C07284=1024.392,-31.797,405.502,166.984,47.714,158.740
C07285=1024.386,-32.047,405.514,166.981,47.718,158.740
C07286=1024.380,-32.296,405.527,166.978,47.721,158.740
C07287=1024.374,-32.546,405.540,166.975,47.724,158.741
C07288=1024.368,-32.796,405.553,166.973,47.727,158.741
C07289=1024.362,-33.046,405.565,166.970,47.731,158.741
C07290=1024.356,-33.295,405.578,166.967,47.734,158.741
C07291=1024.350,-33.545,405.590,166.964,47.737,158.741
C07292=1024.344,-33.794,405.603,166.961,47.740,158.742
C07293=1024.338,-34.044,405.615,166.958,47.744,158.742
C07294=1024.332,-34.293,405.628,166.955,47.747,158.742
C07295=1024.326,-34.543,405.641,166.953,47.750,158.742
C07296=1024.320,-34.793,405.653,166.950,47.753,158.742
C07297=1024.314,-35.043,405.666,166.947,47.757,158.743
C07298=1024.308,-35.292,405.679,166.945,47.760,158.743
C07299=1024.303,-35.541,405.691,166.942,47.763,158.743
C07300=1024.296,-35.791,405.703,166.938,47.766,158.743
C07301=1024.290,-36.040,405.716,166.935,47.770,158.743
C07302=1024.284,-36.290,405.729,166.933,47.772,158.744
C07303=1024.278,-36.570,405.743,166.930,47.776,158.744
C07304=1024.272,-36.849,405.757,166.926,47.780,158.744
C07305=1024.265,-37.129,405.770,166.923,47.784,158.744
C07306=1024.258,-37.408,405.785,166.920,47.787,158.745
C07307=1024.252,-37.658,405.797,166.917,47.791,158.745
C07308=1024.246,-37.908,405.810,166.915,47.793,158.745
C07309=1024.241,-38.157,405.822,166.912,47.797,158.745
C07310=1024.234,-38.407,405.834,166.908,47.800,158.745
C07311=1024.228,-38.656,405.847,166.905,47.803,158.745
C07312=1024.222,-38.906,405.860,166.903,47.807,158.746
C07313=1024.216,-39.156,405.872,166.900,47.810,158.746
C07314=1024.211,-39.405,405.885,166.897,47.813,158.746
C07315=1024.204,-39.654,405.897,166.894,47.816,158.746
C07316=1024.198,-39.904,405.909,166.892,47.820,158.747
C07317=1024.193,-40.155,405.921,166.889,47.823,158.747
C07318=1024.187,-40.404,405.933,166.886,47.826,158.747
C07319=1024.181,-40.654,405.945,166.883,47.830,158.747
C07320=1024.175,-40.903,405.958,166.880,47.833,158.747
C07321=1024.168,-41.153,405.970,166.877,47.836,158.748
C07322=1024.163,-41.402,405.982,166.874,47.840,158.748
C07323=1024.156,-41.652,405.994,166.871,47.843,158.748
C07324=1024.151,-41.902,406.006,166.868,47.846,158.748
C07325=1024.145,-42.152,406.019,166.866,47.850,158.748
C07326=1024.139,-42.400,406.031,166.863,47.853,158.749
C07327=1024.133,-42.650,406.043,166.860,47.856,158.749
C07328=1024.126,-42.900,406.054,166.857,47.859,158.749
C07329=1024.121,-43.150,406.067,166.854,47.863,158.749
C07330=1024.115,-43.400,406.079,166.852,47.866,158.749
C07331=1024.108,-43.649,406.091,166.848,47.869,158.750
C07332=1024.103,-43.899,406.104,166.845,47.873,158.750
C07333=1024.097,-44.148,406.115,166.842,47.876,158.750
C07334=1024.091,-44.398,406.128,166.839,47.879,158.750
C07335=1024.085,-44.648,406.140,166.837,47.882,158.750
C07336=1024.079,-44.897,406.151,166.834,47.886,158.751
C07337=1024.073,-45.147,406.164,166.831,47.889,158.751
C07338=1024.067,-45.396,406.175,166.828,47.892,158.751
C07339=1024.061,-45.646,406.188,166.825,47.895,158.751
C07340=1024.055,-45.896,406.200,166.823,47.899,158.751
C07341=1024.049,-46.145,406.211,166.819,47.902,158.752
C07342=1024.044,-46.395,406.224,166.816,47.905,158.752
C07343=1024.037,-46.645,406.236,166.813,47.909,158.752
C07344=1024.032,-46.894,406.247,166.811,47.912,158.752
C07345=1024.026,-47.144,406.260,166.808,47.915,158.752
C07346=1024.020,-47.393,406.271,166.805,47.918,158.753
C07347=1024.014,-47.643,406.284,166.802,47.922,158.753
C07348=1024.008,-47.893,406.295,166.799,47.925,158.753
C07349=1024.002,-48.142,406.307,166.797,47.928,158.753
C07350=1023.996,-48.392,406.320,166.793,47.932,158.753
C07351=1023.991,-48.642,406.331,166.790,47.935,158.753
C07352=1023.985,-48.892,406.343,166.787,47.938,158.754
C07353=1023.978,-49.141,406.355,166.785,47.941,158.754
C07354=1023.973,-49.391,406.367,166.782,47.945,158.754
C07355=1023.967,-49.641,406.379,166.779,47.948,158.754
C07356=1023.961,-49.890,406.391,166.776,47.951,158.754
C07357=1023.956,-50.140,406.403,166.773,47.954,158.755
C07358=1023.950,-50.389,406.414,166.770,47.957,158.755
C07359=1023.944,-50.639,406.427,166.767,47.961,158.755
C07360=1023.938,-50.889,406.438,166.764,47.964,158.755
C07361=1023.931,-51.138,406.450,166.761,47.967,158.755
C07362=1023.926,-51.389,406.462,166.758,47.971,158.756
C07363=1023.920,-51.637,406.473,166.755,47.974,158.756
C07364=1023.913,-51.888,406.484,166.753,47.978,158.756
C07365=1023.908,-52.137,406.495,166.750,47.981,158.756
C07366=1023.901,-52.387,406.507,166.747,47.984,158.756
C07367=1023.894,-52.666,406.520,166.743,47.988,158.757
C07368=1023.887,-52.947,406.533,166.740,47.992,158.757
C07369=1023.881,-53.227,406.546,166.737,47.996,158.757
C07370=1023.875,-53.507,406.559,166.733,48.000,158.757
C07371=1023.869,-53.756,406.570,166.730,48.004,158.757
C07372=1023.862,-54.006,406.582,166.727,48.007,158.758
C07373=1023.856,-54.255,406.593,166.725,48.010,158.758
C07374=1023.850,-54.505,406.605,166.722,48.013,158.758
C07375=1023.844,-54.755,406.615,166.719,48.017,158.758
C07376=1023.838,-55.005,406.628,166.716,48.021,158.759
C07377=1023.833,-55.254,406.639,166.713,48.024,158.759
C07378=1023.826,-55.504,406.650,166.710,48.028,158.759
C07379=1023.820,-55.753,406.662,166.706,48.031,158.759
C07380=1023.814,-56.003,406.673,166.704,48.035,158.759
C07381=1023.809,-56.253,406.684,166.700,48.038,158.760
C07382=1023.803,-56.502,406.696,166.698,48.041,158.760
C07383=1023.796,-56.752,406.707,166.695,48.045,158.760
C07384=1023.791,-57.002,406.718,166.692,48.048,158.760
C07385=1023.784,-57.251,406.730,166.689,48.052,158.760
C07386=1023.778,-57.501,406.741,166.686,48.055,158.761
C07387=1023.773,-57.751,406.753,166.683,48.058,158.761
C07388=1023.767,-58.001,406.764,166.680,48.062,158.761
C07389=1023.761,-58.250,406.775,166.677,48.065,158.761
C07390=1023.755,-58.500,406.787,166.674,48.068,158.761
C07391=1023.749,-58.749,406.797,166.672,48.072,158.762
C07392=1023.742,-58.999,406.809,166.669,48.075,158.762
C07393=1023.737,-59.249,406.820,166.666,48.079,158.762
C07394=1023.731,-59.498,406.832,166.663,48.082,158.762
C07395=1023.725,-59.748,406.843,166.659,48.085,158.762
C07396=1023.719,-59.998,406.854,166.656,48.089,158.763
C07397=1023.714,-60.247,406.865,166.653,48.092,158.763
C07398=1023.707,-60.497,406.876,166.650,48.096,158.763
C07399=1023.701,-60.746,406.888,166.647,48.099,158.763
C07400=1023.696,-60.996,406.899,166.645,48.102,158.763
C07401=1023.690,-61.246,406.910,166.642,48.106,158.764
C07402=1023.684,-61.496,406.921,166.639,48.109,158.764
C07403=1023.678,-61.745,406.932,166.636,48.113,158.764
C07404=1023.672,-61.995,406.943,166.633,48.116,158.764
C07405=1023.666,-62.245,406.954,166.629,48.119,158.764
C07406=1023.660,-62.494,406.966,166.627,48.123,158.764
C07407=1023.655,-62.744,406.978,166.623,48.126,158.765
C07408=1023.649,-62.994,406.988,166.620,48.129,158.765
C07409=1023.643,-63.243,406.999,166.618,48.133,158.765
C07410=1023.637,-63.494,407.011,166.615,48.136,158.765
C07411=1023.631,-63.743,407.021,166.612,48.139,158.765
C07412=1023.625,-63.992,407.032,166.609,48.143,158.765
C07413=1023.620,-64.242,407.043,166.606,48.146,158.766
C07414=1023.614,-64.492,407.055,166.603,48.150,158.766
C07415=1023.608,-64.742,407.066,166.600,48.153,158.766
C07416=1023.603,-64.991,407.077,166.596,48.156,158.766
C07417=1023.597,-65.241,407.088,166.595,48.160,158.767
C07418=1023.590,-65.491,407.099,166.591,48.163,158.767
C07419=1023.585,-65.741,407.110,166.588,48.166,158.767
C07420=1023.579,-65.990,407.121,166.585,48.169,158.767
C07421=1023.573,-66.240,407.132,166.582,48.173,158.767
C07422=1023.568,-66.489,407.143,166.579,48.176,158.767
C07423=1023.562,-66.740,407.154,166.576,48.180,158.767
C07424=1023.556,-66.989,407.165,166.573,48.183,158.768
C07425=1023.550,-67.239,407.176,166.571,48.186,158.768
C07426=1023.545,-67.488,407.187,166.568,48.190,158.768
C07427=1023.539,-67.738,407.198,166.564,48.193,158.768
C07428=1023.533,-67.988,407.209,166.561,48.196,158.768
C07429=1023.527,-68.237,407.220,166.558,48.200,158.769
C07430=1023.521,-68.487,407.231,166.555,48.203,158.769
C07431=1023.516,-68.768,407.243,166.552,48.206,158.769
C07432=1023.508,-69.049,407.256,166.549,48.210,158.769
C07433=1023.502,-69.330,407.267,166.545,48.214,158.769
C07434=1023.496,-69.612,407.280,166.542,48.218,158.769
C07435=1023.490,-69.861,407.291,166.539,48.221,158.770
C07436=1023.484,-70.111,407.302,166.536,48.225,158.770
C07437=1023.479,-70.360,407.313,166.533,48.228,158.770
C07438=1023.473,-70.610,407.324,166.530,48.231,158.770
C07439=1023.467,-70.859,407.334,166.528,48.234,158.770
C07440=1023.462,-71.109,407.345,166.524,48.237,158.770
C07441=1023.456,-71.359,407.356,166.522,48.241,158.771
C07442=1023.450,-71.609,407.367,166.518,48.244,158.771
C07443=1023.444,-71.859,407.378,166.515,48.247,158.771
C07444=1023.439,-72.108,407.389,166.512,48.251,158.771
C07445=1023.433,-72.358,407.400,166.509,48.254,158.771
C07446=1023.428,-72.608,407.410,166.506,48.257,158.771
C07447=1023.422,-72.858,407.421,166.504,48.261,158.772
C07448=1023.416,-73.107,407.432,166.501,48.264,158.772
C07449=1023.411,-73.356,407.443,166.497,48.267,158.772
C07450=1023.405,-73.606,407.454,166.494,48.270,158.772
C07451=1023.399,-73.856,407.464,166.491,48.274,158.772
C07452=1023.394,-74.106,407.475,166.488,48.277,158.772
C07453=1023.388,-74.355,407.486,166.485,48.281,158.773
C07454=1023.383,-74.605,407.496,166.483,48.284,158.773
C07455=1023.377,-74.855,407.507,166.480,48.287,158.773
C07456=1023.371,-75.105,407.517,166.477,48.291,158.773
C07457=1023.365,-75.355,407.528,166.474,48.294,158.773
C07458=1023.359,-75.604,407.538,166.470,48.297,158.773
C07459=1023.353,-75.854,407.548,166.468,48.301,158.774
C07460=1023.347,-76.104,407.559,166.464,48.304,158.774
C07461=1023.342,-76.354,407.569,166.461,48.307,158.774
C07462=1023.336,-76.603,407.580,166.458,48.311,158.774
C07463=1023.330,-76.853,407.590,166.455,48.315,158.774
C07464=1023.324,-77.103,407.601,166.452,48.318,158.774
C07465=1023.319,-77.353,407.611,166.449,48.322,158.775
C07466=1023.313,-77.602,407.622,166.446,48.325,158.775
C07467=1023.307,-77.852,407.631,166.443,48.328,158.775
C07468=1023.301,-78.102,407.642,166.440,48.332,158.775
C07469=1023.296,-78.352,407.652,166.437,48.335,158.775
C07470=1023.290,-78.601,407.663,166.434,48.338,158.775
C07471=1023.285,-78.851,407.673,166.431,48.342,158.776
C07472=1023.279,-79.100,407.683,166.429,48.345,158.776
C07473=1023.273,-79.350,407.694,166.425,48.349,158.776
C07474=1023.268,-79.599,407.704,166.422,48.352,158.776
C07475=1023.262,-79.849,407.715,166.419,48.356,158.776
C07476=1023.256,-80.099,407.725,166.416,48.359,158.777
C07477=1023.250,-80.349,407.735,166.413,48.362,158.777
C07478=1023.245,-80.599,407.745,166.410,48.366,158.777
C07479=1023.238,-80.848,407.756,166.407,48.369,158.777
C07480=1023.233,-81.098,407.766,166.404,48.373,158.777
C07481=1023.227,-81.348,407.775,166.401,48.376,158.777
C07482=1023.221,-81.597,407.786,166.398,48.380,158.778
C07483=1023.215,-81.847,407.796,166.395,48.383,158.778
C07484=1023.209,-82.097,407.806,166.392,48.387,158.778
C07485=1023.203,-82.347,407.815,166.389,48.391,158.778
C07486=1023.197,-82.597,407.826,166.386,48.395,158.779
C07487=1023.192,-82.846,407.835,166.383,48.398,158.779
C07488=1023.186,-83.096,407.846,166.380,48.402,158.779
C07489=1023.180,-83.346,407.855,166.377,48.405,158.779
C07490=1023.175,-83.595,407.866,166.374,48.408,158.779
C07491=1023.168,-83.845,407.876,166.371,48.412,158.779
C07492=1023.163,-84.095,407.886,166.368,48.415,158.780
C07493=1023.157,-84.345,407.895,166.365,48.419,158.780
C07494=1023.151,-84.595,407.906,166.362,48.422,158.780
C07495=1023.145,-84.877,407.917,166.358,48.427,158.780
C07496=1023.138,-85.161,407.928,166.354,48.431,158.780
C07497=1023.132,-85.443,407.940,166.351,48.435,158.781
C07498=1023.125,-85.727,407.951,166.347,48.439,158.781
C07499=1023.119,-85.977,407.960,166.344,48.442,158.781
C07500=1023.114,-86.227,407.970,166.341,48.446,158.781
C07501=1023.108,-86.476,407.980,166.338,48.449,158.781
C07502=1023.103,-86.726,407.990,166.335,48.453,158.781
C07503=1023.096,-86.975,408.000,166.332,48.457,158.782
C07504=1023.091,-87.225,408.010,166.329,48.460,158.782
C07505=1023.084,-87.475,408.020,166.326,48.464,158.782
C07506=1023.080,-87.725,408.030,166.323,48.467,158.782
C07507=1023.073,-87.974,408.039,166.320,48.470,158.782
C07508=1023.068,-88.225,408.049,166.317,48.474,158.783
C07509=1023.062,-88.474,408.059,166.314,48.477,158.783
C07510=1023.057,-88.724,408.069,166.311,48.481,158.783
C07511=1023.051,-88.974,408.078,166.307,48.484,158.783
C07512=1023.045,-89.224,408.088,166.304,48.488,158.783
C07513=1023.039,-89.473,408.098,166.301,48.492,158.783
C07514=1023.034,-89.723,408.108,166.298,48.495,158.784
C07515=1023.028,-89.973,408.117,166.295,48.498,158.784
C07516=1023.023,-90.223,408.128,166.292,48.502,158.784
C07517=1023.017,-90.472,408.137,166.289,48.505,158.784
C07518=1023.012,-90.722,408.147,166.286,48.509,158.784
C07519=1023.006,-90.972,408.156,166.283,48.512,158.784
C07520=1022.999,-91.222,408.166,166.280,48.516,158.784
C07521=1022.995,-91.471,408.176,166.277,48.520,158.785
C07522=1022.988,-91.721,408.185,166.274,48.523,158.785
C07523=1022.983,-91.971,408.196,166.271,48.526,158.785
C07524=1022.977,-92.220,408.205,166.269,48.530,158.785
C07525=1022.972,-92.470,408.215,166.266,48.533,158.785
C07526=1022.966,-92.720,408.224,166.263,48.536,158.786
C07527=1022.961,-92.969,408.234,166.260,48.540,158.786
C07528=1022.955,-93.219,408.244,166.257,48.543,158.786
C07529=1022.949,-93.469,408.254,166.253,48.547,158.786
C07530=1022.944,-93.718,408.263,166.251,48.551,158.786
C07531=1022.938,-93.969,408.272,166.247,48.554,158.786
C07532=1022.933,-94.218,408.282,166.244,48.557,158.787
C07533=1022.927,-94.468,408.291,166.241,48.561,158.787
C07534=1022.922,-94.718,408.302,166.238,48.564,158.787
C07535=1022.916,-94.967,408.311,166.235,48.567,158.787
C07536=1022.911,-95.217,408.321,166.232,48.571,158.787
C07537=1022.905,-95.466,408.330,166.229,48.575,158.787
C07538=1022.900,-95.717,408.340,166.226,48.578,158.787
C07539=1022.894,-95.967,408.349,166.223,48.582,158.788
C07540=1022.888,-96.216,408.358,166.220,48.585,158.788
C07541=1022.883,-96.466,408.369,166.217,48.588,158.788
C07542=1022.877,-96.715,408.378,166.213,48.591,158.788
C07543=1022.872,-96.966,408.387,166.211,48.595,158.788
C07544=1022.866,-97.215,408.396,166.207,48.599,158.788
C07545=1022.861,-97.465,408.407,166.204,48.602,158.789
C07546=1022.855,-97.714,408.416,166.201,48.606,158.789
C07547=1022.850,-97.965,408.425,166.198,48.609,158.789
C07548=1022.843,-98.214,408.434,166.195,48.612,158.789
C07549=1022.839,-98.464,408.444,166.192,48.616,158.789
C07550=1022.833,-98.714,408.453,166.189,48.620,158.789
C07551=1022.827,-98.963,408.462,166.186,48.623,158.790
C07552=1022.821,-99.213,408.472,166.183,48.627,158.790
C07553=1022.816,-99.463,408.480,166.180,48.631,158.790
C07554=1022.809,-99.713,408.490,166.177,48.634,158.790
C07555=1022.805,-99.963,408.499,166.174,48.638,158.790
C07556=1022.799,-100.212,408.508,166.171,48.641,158.791
C07557=1022.793,-100.462,408.517,166.168,48.645,158.791
C07558=1022.787,-100.712,408.526,166.165,48.648,158.791
C07559=1022.781,-100.997,408.538,166.161,48.653,158.791
C07560=1022.775,-101.282,408.547,166.157,48.657,158.791
C07561=1022.769,-101.568,408.558,166.154,48.661,158.791
C07562=1022.761,-101.853,408.568,166.151,48.665,158.792
C07563=1022.757,-102.103,408.577,166.147,48.668,158.792
C07564=1022.751,-102.353,408.587,166.145,48.672,158.792
C07565=1022.745,-102.602,408.595,166.141,48.675,158.792
C07566=1022.739,-102.852,408.605,166.139,48.679,158.792
C07567=1022.734,-103.102,408.613,166.135,48.683,158.792
C07568=1022.728,-103.351,408.623,166.132,48.686,158.793
C07569=1022.723,-103.602,408.631,166.129,48.690,158.793
C07570=1022.718,-103.851,408.641,166.126,48.693,158.793
C07571=1022.712,-104.101,408.650,166.123,48.697,158.793
C07572=1022.706,-104.350,408.659,166.120,48.700,158.793
C07573=1022.701,-104.600,408.668,166.117,48.704,158.794
C07574=1022.695,-104.850,408.677,166.114,48.708,158.794
C07575=1022.690,-105.100,408.686,166.111,48.711,158.794
C07576=1022.684,-105.350,408.695,166.108,48.715,158.794
C07577=1022.678,-105.599,408.704,166.105,48.718,158.794
C07578=1022.673,-105.849,408.712,166.102,48.722,158.794
C07579=1022.667,-106.099,408.723,166.099,48.725,158.795
C07580=1022.662,-106.349,408.731,166.096,48.729,158.795
C07581=1022.656,-106.599,408.740,166.093,48.732,158.795
C07582=1022.651,-106.848,408.749,166.089,48.736,158.795
C07583=1022.646,-107.098,408.758,166.086,48.740,158.795
C07584=1022.640,-107.348,408.766,166.083,48.743,158.795
C07585=1022.634,-107.598,408.775,166.080,48.747,158.795
C07586=1022.629,-107.847,408.784,166.077,48.750,158.796
C07587=1022.623,-108.098,408.793,166.074,48.754,158.796
C07588=1022.618,-108.347,408.801,166.071,48.758,158.796
C07589=1022.612,-108.596,408.811,166.068,48.762,158.796
C07590=1022.606,-108.847,408.819,166.065,48.765,158.796
C07591=1022.601,-109.097,408.828,166.062,48.769,158.797
C07592=1022.596,-109.346,408.836,166.059,48.772,158.797
C07593=1022.590,-109.597,408.845,166.056,48.776,158.797
C07594=1022.584,-109.845,408.854,166.053,48.779,158.797
C07595=1022.578,-110.095,408.862,166.050,48.783,158.797
C07596=1022.573,-110.345,408.871,166.047,48.787,158.797
C07597=1022.567,-110.595,408.880,166.044,48.791,158.798
C07598=1022.562,-110.845,408.888,166.041,48.794,158.798
C07599=1022.557,-111.095,408.897,166.038,48.798,158.798
C07600=1022.550,-111.345,408.906,166.034,48.801,158.798
C07601=1022.545,-111.594,408.915,166.031,48.805,158.798
C07602=1022.540,-111.844,408.923,166.028,48.809,158.798
C07603=1022.535,-112.094,408.932,166.025,48.812,158.799
C07604=1022.529,-112.344,408.941,166.022,48.816,158.799
C07605=1022.524,-112.594,408.949,166.019,48.820,158.799
C07606=1022.518,-112.844,408.958,166.016,48.823,158.799
C07607=1022.512,-113.093,408.965,166.013,48.827,158.799
C07608=1022.507,-113.343,408.974,166.010,48.830,158.799
C07609=1022.501,-113.592,408.983,166.007,48.834,158.800
C07610=1022.496,-113.842,408.992,166.004,48.837,158.800
C07611=1022.490,-114.092,409.000,166.001,48.841,158.800
C07612=1022.485,-114.342,409.009,165.998,48.845,158.800
C07613=1022.480,-114.591,409.017,165.995,48.848,158.800
C07614=1022.474,-114.842,409.026,165.992,48.852,158.800
C07615=1022.468,-115.091,409.034,165.989,48.855,158.801
C07616=1022.463,-115.341,409.043,165.986,48.859,158.801
C07617=1022.457,-115.591,409.051,165.983,48.863,158.801
C07618=1022.452,-115.840,409.060,165.979,48.867,158.801
C07619=1022.447,-116.091,409.067,165.976,48.871,158.801
C07620=1022.441,-116.341,409.076,165.973,48.874,158.801
C07621=1022.435,-116.590,409.084,165.970,48.878,158.802
C07622=1022.430,-116.840,409.093,165.967,48.881,158.802
C07623=1022.424,-117.125,409.102,165.964,48.885,158.802
C07624=1022.418,-117.410,409.112,165.960,48.889,158.802
C07625=1022.411,-117.695,409.121,165.956,48.894,158.802
C07626=1022.405,-117.980,409.131,165.953,48.898,158.803
C07627=1022.400,-118.229,409.139,165.951,48.902,158.803
C07628=1022.394,-118.480,409.147,165.946,48.905,158.803
C07629=1022.388,-118.730,409.155,165.944,48.909,158.803
C07630=1022.383,-118.980,409.164,165.940,48.913,158.803
C07631=1022.378,-119.229,409.172,165.938,48.917,158.803
C07632=1022.372,-119.479,409.181,165.934,48.920,158.804
C07633=1022.366,-119.728,409.189,165.932,48.924,158.804
C07634=1022.361,-119.979,409.196,165.928,48.927,158.804
C07635=1022.356,-120.228,409.205,165.926,48.931,158.804
C07636=1022.350,-120.478,409.213,165.922,48.934,158.804
C07637=1022.345,-120.727,409.221,165.920,48.938,158.804
C07638=1022.340,-120.977,409.230,165.917,48.942,158.805
C07639=1022.335,-121.228,409.238,165.914,48.946,158.805
C07640=1022.329,-121.477,409.245,165.911,48.950,158.805
C07641=1022.323,-121.727,409.254,165.908,48.953,158.805
C07642=1022.318,-121.977,409.262,165.905,48.957,158.805
C07643=1022.312,-122.226,409.270,165.902,48.960,158.806
C07644=1022.307,-122.476,409.278,165.898,48.964,158.806
C07645=1022.302,-122.726,409.287,165.895,48.968,158.806
C07646=1022.296,-122.976,409.294,165.892,48.972,158.806
C07647=1022.291,-123.226,409.302,165.889,48.975,158.806
C07648=1022.286,-123.475,409.311,165.886,48.979,158.806
C07649=1022.280,-123.725,409.318,165.883,48.982,158.806
C07650=1022.275,-123.975,409.326,165.880,48.986,158.807
C07651=1022.269,-124.225,409.335,165.877,48.989,158.807
C07652=1022.264,-124.475,409.342,165.874,48.993,158.807
C07653=1022.259,-124.724,409.350,165.871,48.997,158.807
C07654=1022.253,-124.975,409.358,165.868,49.001,158.807
C07655=1022.248,-125.224,409.366,165.865,49.004,158.807
C07656=1022.242,-125.474,409.375,165.862,49.008,158.808
C07657=1022.237,-125.724,409.382,165.859,49.012,158.808
C07658=1022.231,-125.974,409.390,165.855,49.016,158.808
C07659=1022.226,-126.224,409.397,165.852,49.020,158.808
C07660=1022.220,-126.473,409.406,165.849,49.023,158.808
C07661=1022.215,-126.723,409.413,165.846,49.027,158.809
C07662=1022.209,-126.973,409.422,165.843,49.031,158.809
C07663=1022.204,-127.223,409.429,165.840,49.034,158.809
C07664=1022.198,-127.473,409.437,165.837,49.038,158.809
C07665=1022.193,-127.723,409.444,165.834,49.041,158.809
C07666=1022.188,-127.972,409.453,165.831,49.045,158.809
C07667=1022.183,-128.222,409.461,165.828,49.049,158.810
C07668=1022.178,-128.471,409.469,165.825,49.051,158.809
C07669=1022.174,-128.721,409.479,165.822,49.054,158.809
C07670=1022.170,-128.971,409.489,165.820,49.056,158.809
C07671=1022.168,-129.220,409.500,165.817,49.057,158.809
C07672=1022.165,-129.469,409.510,165.815,49.058,158.809
C07673=1022.163,-129.719,409.522,165.812,49.058,158.809
C07674=1022.161,-129.969,409.535,165.809,49.058,158.808
C07675=1022.160,-130.219,409.547,165.807,49.057,158.808
C07676=1022.160,-130.469,409.561,165.805,49.056,158.807
C07677=1022.159,-130.719,409.575,165.803,49.054,158.807
C07678=1022.160,-130.968,409.590,165.801,49.052,158.806
C07679=1022.160,-131.219,409.604,165.798,49.050,158.805
C07680=1022.162,-131.469,409.621,165.797,49.046,158.804
C07681=1022.164,-131.718,409.637,165.795,49.042,158.803
C07682=1022.166,-131.967,409.654,165.793,49.038,158.802
C07683=1022.170,-132.218,409.671,165.792,49.033,158.801
C07684=1022.172,-132.467,409.690,165.790,49.028,158.800
C07685=1022.177,-132.717,409.708,165.788,49.022,158.799
C07686=1022.181,-132.966,409.727,165.786,49.016,158.798
///RCONF 1,0,0,0,1,0,0,0,0,0,0,0,0,0,0,0,0,0,0,0,0,0,0,0
C07687=1021.894,-132.993,409.379,165.740,49.314,158.841
C07688=1021.889,-132.743,409.360,165.742,49.320,158.842
C07689=1021.885,-132.493,409.340,165.743,49.325,158.843
C07690=1021.882,-132.243,409.323,165.744,49.331,158.845
C07691=1021.880,-131.993,409.305,165.746,49.336,158.846
C07692=1021.877,-131.744,409.288,165.748,49.340,158.847
///RCONF 1,0,0,0,0,0,0,0,0,0,0,0,0,0,0,0,0,0,0,0,0,0,0,0
C07693=1021.875,-131.494,409.272,165.750,49.344,158.848
C07694=1021.874,-131.244,409.256,165.752,49.346,158.848
C07695=1021.873,-130.994,409.240,165.753,49.349,158.849
C07696=1021.873,-130.744,409.225,165.756,49.352,158.850
C07697=1021.872,-130.495,409.212,165.758,49.354,158.850
C07698=1021.874,-130.245,409.199,165.761,49.355,158.851
C07699=1021.874,-129.995,409.185,165.763,49.355,158.851
C07700=1021.876,-129.746,409.173,165.765,49.355,158.852
C07701=1021.878,-129.496,409.162,165.768,49.355,158.852
C07702=1021.880,-129.246,409.151,165.770,49.355,158.852
C07703=1021.883,-128.996,409.140,165.773,49.353,158.853
C07704=1021.887,-128.747,409.130,165.775,49.351,158.853
C07705=1021.891,-128.497,409.120,165.779,49.349,158.853
C07706=1021.895,-128.248,409.112,165.781,49.346,158.853
C07707=1021.901,-127.998,409.103,165.784,49.342,158.853
C07708=1021.905,-127.748,409.095,165.787,49.339,158.853
C07709=1021.911,-127.499,409.088,165.790,49.335,158.852
C07710=1021.916,-127.249,409.080,165.793,49.331,158.852
C07711=1021.922,-127.000,409.072,165.797,49.328,158.852
C07712=1021.927,-126.749,409.065,165.800,49.323,158.852
C07713=1021.933,-126.500,409.057,165.803,49.319,158.852
C07714=1021.938,-126.250,409.049,165.806,49.316,158.852
C07715=1021.944,-126.000,409.041,165.809,49.312,158.851
C07716=1021.949,-125.750,409.033,165.812,49.309,158.851
C07717=1021.955,-125.500,409.025,165.815,49.305,158.851
C07718=1021.960,-125.250,409.018,165.817,49.301,158.851
C07719=1021.966,-125.001,409.010,165.821,49.297,158.851
C07720=1021.971,-124.750,409.002,165.824,49.293,158.850
C07721=1021.977,-124.501,408.994,165.827,49.289,158.850
C07722=1021.981,-124.252,408.986,165.830,49.286,158.850
C07723=1021.986,-124.002,408.978,165.833,49.282,158.850
C07724=1021.992,-123.752,408.970,165.836,49.278,158.850
C07725=1021.997,-123.502,408.962,165.839,49.274,158.850
C07726=1022.003,-123.252,408.954,165.842,49.271,158.849
C07727=1022.009,-123.003,408.946,165.845,49.267,158.849
C07728=1022.013,-122.752,408.938,165.848,49.263,158.849
C07729=1022.019,-122.503,408.930,165.852,49.260,158.849
C07730=1022.025,-122.253,408.922,165.855,49.256,158.849
C07731=1022.030,-122.003,408.914,165.858,49.252,158.849
C07732=1022.035,-121.753,408.906,165.861,49.248,158.848
C07733=1022.040,-121.503,408.897,165.864,49.245,158.848
C07734=1022.046,-121.254,408.889,165.867,49.241,158.848
C07735=1022.051,-121.004,408.882,165.869,49.237,158.848
C07736=1022.056,-120.754,408.873,165.872,49.234,158.848
C07737=1022.062,-120.505,408.865,165.875,49.230,158.847
C07738=1022.068,-120.255,408.857,165.878,49.226,158.847
C07739=1022.073,-120.005,408.849,165.882,49.222,158.847
C07740=1022.079,-119.754,408.841,165.885,49.219,158.847
C07741=1022.085,-119.505,408.832,165.888,49.215,158.847
C07742=1022.090,-119.255,408.824,165.891,49.211,158.847
C07743=1022.095,-119.005,408.816,165.894,49.207,158.847
C07744=1022.101,-118.755,408.808,165.897,49.203,158.846
C07745=1022.106,-118.506,408.800,165.900,49.200,158.846
C07746=1022.111,-118.256,408.791,165.903,49.196,158.846
C07747=1022.117,-118.006,408.783,165.906,49.192,158.846
C07748=1022.123,-117.721,408.773,165.910,49.188,158.846
C07749=1022.129,-117.436,408.764,165.913,49.183,158.845
C07750=1022.135,-117.151,408.755,165.916,49.179,158.845
C07751=1022.141,-116.866,408.745,165.920,49.175,158.845
C07752=1022.147,-116.617,408.737,165.923,49.172,158.845
C07753=1022.153,-116.367,408.729,165.926,49.168,158.845
C07754=1022.158,-116.117,408.720,165.929,49.164,158.844
C07755=1022.164,-115.867,408.711,165.933,49.160,158.844
C07756=1022.169,-115.617,408.703,165.936,49.156,158.844
C07757=1022.175,-115.368,408.695,165.939,49.153,158.844
C07758=1022.180,-115.118,408.687,165.942,49.149,158.844
C07759=1022.185,-114.868,408.678,165.945,49.146,158.844
C07760=1022.191,-114.619,408.670,165.948,49.142,158.843
C07761=1022.197,-114.368,408.661,165.950,49.138,158.843
C07762=1022.203,-114.119,408.653,165.954,49.134,158.843
C07763=1022.208,-113.869,408.644,165.956,49.130,158.843
C07764=1022.213,-113.619,408.636,165.961,49.127,158.843
C07765=1022.218,-113.370,408.627,165.963,49.123,158.843
C07766=1022.224,-113.119,408.619,165.967,49.119,158.843
C07767=1022.230,-112.869,408.610,165.969,49.115,158.842
C07768=1022.235,-112.620,408.602,165.973,49.112,158.842
C07769=1022.240,-112.370,408.593,165.975,49.108,158.842
C07770=1022.245,-112.120,408.585,165.978,49.105,158.842
C07771=1022.251,-111.870,408.576,165.981,49.101,158.842
C07772=1022.256,-111.620,408.567,165.984,49.098,158.841
C07773=1022.262,-111.370,408.559,165.987,49.094,158.841
C07774=1022.268,-111.121,408.551,165.990,49.090,158.841
C07775=1022.274,-110.871,408.541,165.994,49.086,158.841
C07776=1022.279,-110.622,408.533,165.997,49.082,158.841
C07777=1022.284,-110.372,408.524,166.000,49.079,158.841
C07778=1022.290,-110.122,408.516,166.003,49.075,158.840
C07779=1022.296,-109.872,408.507,166.006,49.071,158.840
C07780=1022.301,-109.622,408.498,166.009,49.067,158.840
C07781=1022.306,-109.373,408.489,166.012,49.064,158.840
C07782=1022.312,-109.123,408.481,166.015,49.060,158.840
C07783=1022.318,-108.873,408.472,166.018,49.056,158.839
C07784=1022.323,-108.623,408.463,166.021,49.053,158.839
C07785=1022.328,-108.373,408.455,166.025,49.049,158.839
C07786=1022.334,-108.123,408.445,166.028,49.045,158.839
C07787=1022.339,-107.874,408.437,166.031,49.041,158.839
C07788=1022.345,-107.624,408.428,166.034,49.038,158.839
C07789=1022.351,-107.374,408.420,166.037,49.034,158.838
C07790=1022.356,-107.125,408.410,166.040,49.031,158.838
C07791=1022.361,-106.875,408.402,166.043,49.027,158.838
C07792=1022.367,-106.624,408.393,166.046,49.023,158.838
C07793=1022.373,-106.375,408.385,166.049,49.019,158.838
C07794=1022.378,-106.126,408.375,166.052,49.016,158.838
C07795=1022.384,-105.875,408.367,166.054,49.012,158.837
C07796=1022.390,-105.626,408.357,166.059,49.009,158.837
C07797=1022.395,-105.376,408.349,166.061,49.005,158.837
C07798=1022.401,-105.126,408.340,166.065,49.001,158.837
C07799=1022.406,-104.877,408.331,166.067,48.997,158.837
C07800=1022.411,-104.626,408.321,166.071,48.994,158.837
C07801=1022.417,-104.376,408.313,166.073,48.990,158.836
C07802=1022.422,-104.127,408.304,166.077,48.987,158.836
C07803=1022.428,-103.877,408.295,166.079,48.983,158.836
C07804=1022.434,-103.628,408.286,166.083,48.980,158.836
C07805=1022.440,-103.377,408.277,166.085,48.976,158.836
C07806=1022.445,-103.128,408.268,166.088,48.972,158.836
C07807=1022.450,-102.879,408.259,166.091,48.968,158.835
C07808=1022.455,-102.628,408.250,166.094,48.965,158.835
C07809=1022.461,-102.379,408.240,166.097,48.961,158.835
C07810=1022.467,-102.128,408.232,166.101,48.957,158.835
C07811=1022.473,-101.879,408.222,166.104,48.954,158.835
C07812=1022.479,-101.593,408.212,166.107,48.950,158.834
C07813=1022.485,-101.309,408.202,166.111,48.945,158.834
C07814=1022.491,-101.023,408.191,166.115,48.941,158.834
C07815=1022.498,-100.738,408.180,166.118,48.937,158.834
C07816=1022.504,-100.489,408.172,166.121,48.934,158.834
C07817=1022.510,-100.239,408.162,166.124,48.930,158.833
C07818=1022.514,-99.989,408.153,166.128,48.926,158.833
C07819=1022.521,-99.739,408.144,166.131,48.922,158.833
C07820=1022.526,-99.490,408.135,166.134,48.919,158.833
C07821=1022.532,-99.239,408.126,166.137,48.915,158.833
C07822=1022.538,-98.990,408.117,166.140,48.912,158.833
C07823=1022.543,-98.740,408.108,166.143,48.908,158.832
C07824=1022.548,-98.490,408.098,166.145,48.904,158.832
C07825=1022.554,-98.241,408.088,166.148,48.900,158.832
C07826=1022.560,-97.991,408.080,166.151,48.896,158.832
C07827=1022.566,-97.741,408.070,166.154,48.893,158.832
C07828=1022.571,-97.492,408.060,166.157,48.889,158.831
C07829=1022.577,-97.241,408.052,166.160,48.886,158.831
C07830=1022.582,-96.992,408.042,166.164,48.883,158.831
C07831=1022.588,-96.742,408.032,166.166,48.879,158.831
C07832=1022.593,-96.493,408.023,166.170,48.875,158.831
C07833=1022.598,-96.242,408.014,166.173,48.872,158.831
C07834=1022.604,-95.993,408.004,166.176,48.868,158.831
C07835=1022.609,-95.743,407.994,166.179,48.865,158.830
C07836=1022.615,-95.493,407.985,166.182,48.862,158.830
C07837=1022.621,-95.244,407.975,166.185,48.858,158.830
C07838=1022.626,-94.993,407.966,166.188,48.854,158.830
C07839=1022.632,-94.744,407.957,166.191,48.851,158.830
C07840=1022.637,-94.494,407.947,166.195,48.847,158.830
C07841=1022.643,-94.245,407.937,166.198,48.844,158.830
C07842=1022.648,-93.995,407.927,166.201,48.840,158.829
C07843=1022.654,-93.745,407.918,166.204,48.836,158.829
C07844=1022.659,-93.495,407.909,166.207,48.833,158.829
C07845=1022.665,-93.245,407.899,166.210,48.829,158.829
C07846=1022.671,-92.996,407.890,166.213,48.826,158.829
C07847=1022.676,-92.746,407.880,166.216,48.822,158.828
C07848=1022.682,-92.496,407.870,166.219,48.819,158.828
C07849=1022.687,-92.247,407.860,166.222,48.815,158.828
C07850=1022.693,-91.997,407.851,166.225,48.812,158.828
C07851=1022.699,-91.747,407.841,166.228,48.808,158.828
C07852=1022.704,-91.498,407.831,166.231,48.804,158.828
C07853=1022.710,-91.248,407.821,166.234,48.801,158.828
C07854=1022.716,-90.998,407.812,166.237,48.797,158.827
C07855=1022.721,-90.749,407.802,166.240,48.794,158.827
C07856=1022.727,-90.498,407.793,166.243,48.790,158.827
C07857=1022.732,-90.248,407.783,166.246,48.787,158.827
C07858=1022.738,-89.999,407.774,166.249,48.783,158.827
C07859=1022.744,-89.749,407.764,166.252,48.779,158.826
C07860=1022.749,-89.499,407.754,166.255,48.776,158.826
C07861=1022.755,-89.249,407.744,166.258,48.772,158.826
C07862=1022.760,-89.000,407.735,166.261,48.769,158.826
C07863=1022.766,-88.750,407.725,166.264,48.765,158.826
C07864=1022.772,-88.501,407.714,166.267,48.762,158.826
C07865=1022.778,-88.251,407.705,166.270,48.758,158.825
C07866=1022.783,-88.002,407.695,166.273,48.754,158.825
C07867=1022.789,-87.752,407.685,166.276,48.751,158.825
C07868=1022.795,-87.502,407.675,166.279,48.747,158.825
C07869=1022.801,-87.252,407.666,166.282,48.744,158.825
C07870=1022.806,-87.002,407.656,166.286,48.740,158.824
C07871=1022.812,-86.753,407.646,166.289,48.737,158.824
C07872=1022.817,-86.502,407.636,166.292,48.733,158.824
C07873=1022.823,-86.253,407.626,166.295,48.729,158.824
C07874=1022.828,-86.003,407.617,166.298,48.725,158.824
C07875=1022.834,-85.753,407.607,166.301,48.722,158.824
C07876=1022.842,-85.470,407.595,166.304,48.718,158.823
C07877=1022.847,-85.187,407.584,166.308,48.714,158.823
C07878=1022.854,-84.904,407.572,166.312,48.710,158.823
C07879=1022.861,-84.621,407.562,166.315,48.706,158.823
C07880=1022.866,-84.371,407.552,166.318,48.702,158.822
C07881=1022.872,-84.121,407.542,166.321,48.699,158.822
C07882=1022.878,-83.871,407.532,166.324,48.695,158.822
C07883=1022.884,-83.622,407.522,166.327,48.691,158.822
C07884=1022.890,-83.372,407.512,166.329,48.687,158.822
C07885=1022.895,-83.123,407.502,166.334,48.684,158.822
C07886=1022.901,-82.873,407.492,166.337,48.680,158.821
C07887=1022.907,-82.623,407.483,166.340,48.677,158.821
C07888=1022.912,-82.374,407.472,166.343,48.673,158.821
C07889=1022.919,-82.124,407.462,166.346,48.669,158.821
C07890=1022.924,-81.874,407.452,166.348,48.666,158.821
C07891=1022.930,-81.624,407.442,166.351,48.662,158.820
C07892=1022.936,-81.374,407.432,166.354,48.658,158.820
C07893=1022.942,-81.125,407.422,166.357,48.654,158.820
C07894=1022.947,-80.875,407.412,166.360,48.651,158.820
C07895=1022.953,-80.626,407.402,166.363,48.647,158.820
C07896=1022.959,-80.376,407.392,166.366,48.644,158.819
C07897=1022.965,-80.126,407.382,166.369,48.640,158.819
C07898=1022.971,-79.877,407.371,166.372,48.637,158.819
C07899=1022.976,-79.626,407.361,166.375,48.633,158.819
C07900=1022.982,-79.376,407.351,166.378,48.630,158.819
C07901=1022.988,-79.127,407.341,166.382,48.626,158.819
C07902=1022.994,-78.877,407.331,166.384,48.622,158.818
C07903=1022.999,-78.628,407.320,166.388,48.619,158.818
C07904=1023.005,-78.377,407.309,166.390,48.615,158.818
C07905=1023.010,-78.128,407.299,166.394,48.612,158.818
C07906=1023.017,-77.878,407.289,166.397,48.609,158.818
C07907=1023.022,-77.629,407.278,166.400,48.605,158.817
C07908=1023.028,-77.379,407.268,166.403,48.602,158.817
C07909=1023.034,-77.129,407.257,166.406,48.598,158.817
C07910=1023.040,-76.879,407.248,166.409,48.594,158.817
C07911=1023.045,-76.630,407.237,166.412,48.591,158.817
C07912=1023.051,-76.380,407.227,166.415,48.587,158.816
C07913=1023.057,-76.130,407.216,166.418,48.584,158.816
C07914=1023.062,-75.880,407.205,166.421,48.580,158.816
C07915=1023.069,-75.631,407.195,166.424,48.577,158.816
C07916=1023.074,-75.381,407.185,166.427,48.574,158.816
C07917=1023.080,-75.131,407.174,166.430,48.570,158.816
C07918=1023.085,-74.881,407.164,166.433,48.566,158.815
C07919=1023.091,-74.632,407.153,166.436,48.562,158.815
C07920=1023.097,-74.383,407.143,166.439,48.559,158.815
C07921=1023.103,-74.132,407.133,166.442,48.556,158.815
C07922=1023.108,-73.883,407.121,166.445,48.552,158.815
C07923=1023.114,-73.633,407.110,166.448,48.549,158.815
C07924=1023.119,-73.383,407.100,166.451,48.546,158.814
C07925=1023.125,-73.134,407.089,166.455,48.542,158.814
C07926=1023.130,-72.884,407.078,166.457,48.538,158.814
C07927=1023.136,-72.635,407.068,166.460,48.535,158.814
C07928=1023.142,-72.384,407.057,166.463,48.532,158.814
C07929=1023.147,-72.135,407.047,166.466,48.529,158.814
C07930=1023.153,-71.886,407.036,166.469,48.525,158.813
C07931=1023.159,-71.636,407.025,166.472,48.522,158.813
C07932=1023.164,-71.386,407.015,166.475,48.519,158.813
C07933=1023.169,-71.136,407.003,166.478,48.515,158.813
C07934=1023.175,-70.887,406.992,166.481,48.511,158.813
C07935=1023.181,-70.636,406.981,166.484,48.508,158.813
C07936=1023.187,-70.387,406.970,166.487,48.505,158.812
C07937=1023.193,-70.137,406.959,166.490,48.502,158.812
C07938=1023.198,-69.887,406.949,166.492,48.498,158.812
C07939=1023.204,-69.638,406.938,166.495,48.495,158.812
C07940=1023.211,-69.358,406.926,166.499,48.491,158.812
C07941=1023.217,-69.076,406.913,166.502,48.487,158.812
C07942=1023.223,-68.795,406.902,166.506,48.483,158.811
C07943=1023.230,-68.514,406.889,166.509,48.479,158.811
C07944=1023.235,-68.265,406.878,166.512,48.476,158.811
C07945=1023.242,-68.015,406.867,166.516,48.473,158.811
C07946=1023.247,-67.765,406.856,166.518,48.469,158.811
C07947=1023.252,-67.515,406.845,166.522,48.466,158.810
C07948=1023.258,-67.265,406.834,166.525,48.463,158.810
C07949=1023.264,-67.016,406.824,166.528,48.459,158.810
C07950=1023.269,-66.766,406.813,166.530,48.456,158.810
C07951=1023.276,-66.516,406.801,166.533,48.452,158.810
C07952=1023.281,-66.267,406.791,166.536,48.449,158.809
C07953=1023.287,-66.017,406.780,166.539,48.445,158.809
C07954=1023.293,-65.768,406.769,166.542,48.442,158.809
C07955=1023.299,-65.518,406.758,166.545,48.438,158.809
C07956=1023.304,-65.268,406.746,166.548,48.435,158.809
C07957=1023.310,-65.018,406.735,166.551,48.432,158.809
C07958=1023.316,-64.769,406.724,166.554,48.428,158.808
C07959=1023.321,-64.519,406.714,166.557,48.425,158.808
C07960=1023.328,-64.269,406.702,166.560,48.421,158.808
C07961=1023.334,-64.019,406.691,166.563,48.417,158.808
C07962=1023.339,-63.770,406.681,166.566,48.414,158.808
C07963=1023.345,-63.520,406.670,166.569,48.410,158.807
C07964=1023.351,-63.270,406.658,166.571,48.407,158.807
C07965=1023.356,-63.020,406.647,166.575,48.404,158.807
C07966=1023.362,-62.772,406.635,166.577,48.400,158.807
C07967=1023.368,-62.522,406.624,166.581,48.397,158.807
C07968=1023.375,-62.272,406.613,166.584,48.394,158.807
C07969=1023.380,-62.022,406.602,166.587,48.390,158.806
C07970=1023.386,-61.773,406.591,166.590,48.387,158.806
C07971=1023.392,-61.522,406.580,166.593,48.383,158.806
C07972=1023.397,-61.273,406.569,166.596,48.380,158.806
C07973=1023.403,-61.023,406.558,166.599,48.376,158.806
C07974=1023.409,-60.773,406.547,166.602,48.372,158.805
C07975=1023.415,-60.524,406.536,166.605,48.369,158.805
C07976=1023.421,-60.275,406.524,166.608,48.365,158.805
C07977=1023.428,-60.025,406.513,166.611,48.362,158.805
C07978=1023.433,-59.775,406.501,166.614,48.358,158.804
C07979=1023.438,-59.525,406.491,166.616,48.355,158.804
C07980=1023.445,-59.275,406.479,166.619,48.352,158.804
C07981=1023.451,-59.026,406.468,166.622,48.348,158.804
C07982=1023.456,-58.777,406.457,166.625,48.345,158.804
C07983=1023.463,-58.527,406.446,166.628,48.341,158.803
C07984=1023.468,-58.277,406.434,166.631,48.338,158.803
C07985=1023.473,-58.027,406.423,166.634,48.334,158.803
C07986=1023.480,-57.778,406.411,166.637,48.331,158.803
C07987=1023.486,-57.528,406.400,166.640,48.327,158.803
C07988=1023.492,-57.278,406.389,166.643,48.324,158.802
C07989=1023.498,-57.029,406.378,166.646,48.320,158.802
C07990=1023.503,-56.779,406.366,166.649,48.316,158.802
C07991=1023.510,-56.529,406.355,166.652,48.313,158.802
C07992=1023.515,-56.280,406.344,166.655,48.309,158.802
C07993=1023.522,-56.030,406.333,166.658,48.306,158.802
C07994=1023.528,-55.781,406.321,166.661,48.302,158.801
C07995=1023.534,-55.531,406.310,166.664,48.299,158.801
C07996=1023.539,-55.281,406.298,166.667,48.295,158.801
C07997=1023.545,-55.032,406.287,166.669,48.292,158.801
C07998=1023.551,-54.782,406.276,166.672,48.288,158.800
C07999=1023.557,-54.532,406.265,166.675,48.285,158.800
C08000=1023.564,-54.283,406.253,166.678,48.281,158.800
C08001=1023.570,-54.033,406.242,166.681,48.278,158.800
C08002=1023.575,-53.783,406.230,166.684,48.274,158.799
C08003=1023.581,-53.534,406.218,166.687,48.271,158.799
C08004=1023.588,-53.253,406.206,166.691,48.267,158.799
C08005=1023.595,-52.974,406.193,166.694,48.263,158.799
C08006=1023.602,-52.694,406.180,166.697,48.259,158.799
C08007=1023.608,-52.414,406.167,166.701,48.255,158.798
C08008=1023.615,-52.164,406.156,166.704,48.251,158.798
C08009=1023.621,-51.915,406.145,166.707,48.248,158.798
C08010=1023.627,-51.665,406.133,166.710,48.244,158.798
C08011=1023.632,-51.415,406.121,166.713,48.240,158.797
C08012=1023.639,-51.165,406.110,166.716,48.237,158.797
C08013=1023.645,-50.916,406.098,166.719,48.233,158.797
C08014=1023.651,-50.666,406.087,166.721,48.230,158.797
C08015=1023.656,-50.417,406.075,166.724,48.227,158.797
C08016=1023.662,-50.167,406.062,166.727,48.223,158.796
C08017=1023.668,-49.918,406.052,166.730,48.220,158.796
C08018=1023.674,-49.668,406.039,166.733,48.216,158.796
C08019=1023.680,-49.418,406.028,166.736,48.213,158.796
C08020=1023.685,-49.168,406.016,166.738,48.210,158.796
C08021=1023.692,-48.919,406.004,166.742,48.207,158.796
C08022=1023.697,-48.669,405.992,166.745,48.203,158.795
C08023=1023.703,-48.419,405.980,166.748,48.200,158.795
C08024=1023.709,-48.170,405.968,166.751,48.197,158.795
C08025=1023.715,-47.920,405.956,166.754,48.193,158.795
C08026=1023.721,-47.671,405.945,166.756,48.190,158.794
C08027=1023.727,-47.421,405.932,166.759,48.187,158.794
C08028=1023.733,-47.172,405.920,166.762,48.183,158.794
C08029=1023.738,-46.922,405.909,166.765,48.180,158.794
C08030=1023.744,-46.672,405.896,166.768,48.176,158.794
C08031=1023.750,-46.423,405.884,166.771,48.173,158.793
C08032=1023.756,-46.172,405.873,166.773,48.170,158.793
C08033=1023.762,-45.923,405.861,166.776,48.166,158.793
C08034=1023.768,-45.674,405.848,166.779,48.163,158.793
C08035=1023.774,-45.424,405.836,166.782,48.159,158.793
C08036=1023.779,-45.174,405.825,166.786,48.156,158.793
C08037=1023.785,-44.924,405.812,166.788,48.152,158.792
C08038=1023.792,-44.675,405.800,166.792,48.149,158.792
C08039=1023.797,-44.426,405.788,166.794,48.146,158.792
C08040=1023.803,-44.176,405.776,166.797,48.142,158.792
C08041=1023.810,-43.925,405.764,166.800,48.139,158.791
C08042=1023.815,-43.676,405.752,166.803,48.136,158.791
C08043=1023.821,-43.427,405.740,166.806,48.132,158.791
C08044=1023.827,-43.177,405.728,166.809,48.129,158.791
C08045=1023.833,-42.928,405.716,166.811,48.125,158.790
C08046=1023.839,-42.678,405.704,166.814,48.122,158.790
C08047=1023.845,-42.428,405.692,166.817,48.119,158.790
C08048=1023.851,-42.179,405.680,166.820,48.115,158.790
C08049=1023.857,-41.929,405.668,166.823,48.112,158.790
C08050=1023.863,-41.679,405.655,166.826,48.109,158.790
C08051=1023.869,-41.430,405.643,166.828,48.105,158.789
C08052=1023.875,-41.180,405.631,166.831,48.102,158.789
C08053=1023.881,-40.931,405.619,166.834,48.098,158.789
C08054=1023.887,-40.681,405.606,166.838,48.095,158.789
C08055=1023.893,-40.432,405.594,166.840,48.091,158.788
C08056=1023.899,-40.181,405.583,166.844,48.088,158.788
C08057=1023.905,-39.931,405.570,166.847,48.084,158.788
C08058=1023.911,-39.682,405.558,166.849,48.081,158.788
C08059=1023.917,-39.433,405.546,166.852,48.078,158.788
C08060=1023.923,-39.183,405.534,166.855,48.074,158.787
C08061=1023.929,-38.933,405.521,166.858,48.071,158.787
C08062=1023.935,-38.683,405.509,166.861,48.067,158.787
C08063=1023.941,-38.434,405.497,166.863,48.065,158.787
C08064=1023.947,-38.184,405.484,166.866,48.061,158.786
C08065=1023.952,-37.934,405.472,166.869,48.057,158.786
C08066=1023.959,-37.685,405.459,166.872,48.054,158.786
C08067=1023.964,-37.436,405.446,166.874,48.051,158.786
C08068=1023.970,-37.156,405.433,166.878,48.047,158.786
C08069=1023.977,-36.877,405.419,166.881,48.043,158.785
C08070=1023.984,-36.598,405.405,166.884,48.039,158.785
C08071=1023.990,-36.318,405.391,166.887,48.036,158.785
C08072=1023.997,-36.069,405.378,166.890,48.032,158.785
C08073=1024.003,-35.819,405.366,166.893,48.029,158.785
C08074=1024.009,-35.569,405.353,166.896,48.026,158.784
C08075=1024.015,-35.319,405.341,166.899,48.023,158.784
C08076=1024.020,-35.070,405.328,166.902,48.019,158.784
C08077=1024.026,-34.820,405.316,166.905,48.016,158.784
C08078=1024.032,-34.571,405.303,166.908,48.013,158.784
C08079=1024.038,-34.321,405.290,166.911,48.009,158.783
C08080=1024.044,-34.071,405.277,166.913,48.006,158.783
C08081=1024.051,-33.821,405.265,166.916,48.003,158.783
C08082=1024.056,-33.572,405.253,166.919,47.999,158.783
C08083=1024.062,-33.323,405.240,166.922,47.996,158.783
C08084=1024.068,-33.073,405.227,166.924,47.993,158.782
C08085=1024.074,-32.823,405.215,166.927,47.989,158.782
C08086=1024.080,-32.573,405.202,166.930,47.986,158.782
C08087=1024.086,-32.324,405.189,166.933,47.983,158.782
C08088=1024.092,-32.074,405.177,166.935,47.979,158.781
C08089=1024.098,-31.824,405.164,166.939,47.976,158.781
C08090=1024.103,-31.575,405.152,166.941,47.972,158.781
C08091=1024.110,-31.326,405.139,166.945,47.969,158.781
C08092=1024.116,-31.076,405.127,166.948,47.966,158.781
C08093=1024.122,-30.826,405.114,166.950,47.962,158.780
C08094=1024.128,-30.577,405.101,166.953,47.959,158.780
C08095=1024.134,-30.327,405.088,166.956,47.956,158.780
C08096=1024.140,-30.077,405.076,166.959,47.952,158.780
C08097=1024.146,-29.828,405.062,166.961,47.949,158.779
C08098=1024.152,-29.578,405.050,166.964,47.945,158.779
C08099=1024.158,-29.328,405.037,166.967,47.942,158.779
C08100=1024.164,-29.079,405.024,166.970,47.939,158.779
C08101=1024.170,-28.829,405.011,166.973,47.935,158.778
C08102=1024.177,-28.579,404.999,166.975,47.932,158.778
C08103=1024.183,-28.330,404.986,166.978,47.928,158.778
C08104=1024.189,-28.080,404.974,166.981,47.925,158.778
C08105=1024.195,-27.830,404.961,166.984,47.922,158.778
C08106=1024.200,-27.582,404.948,166.987,47.918,158.777
C08107=1024.206,-27.332,404.936,166.989,47.915,158.777
C08108=1024.212,-27.083,404.922,166.992,47.911,158.777
C08109=1024.218,-26.833,404.909,166.996,47.908,158.777
C08110=1024.224,-26.583,404.896,166.998,47.905,158.776
C08111=1024.230,-26.333,404.883,167.001,47.902,158.776
C08112=1024.236,-26.084,404.870,167.004,47.898,158.776
C08113=1024.242,-25.834,404.858,167.006,47.895,158.776
C08114=1024.248,-25.585,404.844,167.009,47.892,158.776
C08115=1024.254,-25.335,404.830,167.012,47.889,158.775
C08116=1024.259,-25.086,404.818,167.015,47.885,158.775
C08117=1024.266,-24.836,404.805,167.017,47.882,158.775
C08118=1024.272,-24.586,404.792,167.021,47.879,158.775
C08119=1024.278,-24.337,404.779,167.024,47.876,158.775
C08120=1024.283,-24.088,404.765,167.026,47.872,158.774
C08121=1024.289,-23.838,404.752,167.029,47.869,158.774
C08122=1024.295,-23.588,404.739,167.032,47.866,158.774
C08123=1024.301,-23.338,404.727,167.035,47.862,158.774
C08124=1024.308,-23.089,404.713,167.037,47.859,158.773
C08125=1024.314,-22.839,404.699,167.040,47.856,158.773
C08126=1024.320,-22.589,404.686,167.043,47.852,158.773
C08127=1024.326,-22.340,404.673,167.045,47.849,158.773
C08128=1024.332,-22.091,404.660,167.048,47.846,158.773
C08129=1024.338,-21.841,404.647,167.051,47.842,158.772
C08130=1024.343,-21.591,404.634,167.053,47.840,158.772
C08131=1024.350,-21.342,404.620,167.057,47.836,158.772
C08132=1024.356,-21.061,404.606,167.059,47.833,158.772
C08133=1024.363,-20.781,404.591,167.062,47.829,158.771
C08134=1024.370,-20.501,404.576,167.066,47.825,158.771
C08135=1024.377,-20.221,404.561,167.069,47.821,158.771
C08136=1024.383,-19.971,404.548,167.072,47.818,158.771
C08137=1024.388,-19.721,404.535,167.074,47.815,158.770
C08138=1024.394,-19.472,404.522,167.078,47.812,158.770
C08139=1024.401,-19.223,404.508,167.081,47.808,158.770
C08140=1024.407,-18.973,404.495,167.083,47.805,158.770
C08141=1024.413,-18.723,404.482,167.086,47.802,158.769
C08142=1024.419,-18.473,404.468,167.089,47.798,158.769
C08143=1024.425,-18.224,404.455,167.092,47.795,158.769
C08144=1024.431,-17.975,404.442,167.094,47.791,158.769
C08145=1024.437,-17.725,404.429,167.097,47.788,158.768
C08146=1024.443,-17.475,404.415,167.100,47.785,158.768
C08147=1024.449,-17.225,404.402,167.102,47.781,158.768
C08148=1024.456,-16.976,404.388,167.105,47.778,158.768
C08149=1024.462,-16.727,404.375,167.108,47.774,158.767
C08150=1024.468,-16.477,404.363,167.111,47.771,158.767
C08151=1024.473,-16.227,404.349,167.113,47.768,158.767
C08152=1024.480,-15.977,404.335,167.116,47.764,158.767
C08153=1024.486,-15.728,404.322,167.119,47.761,158.767
C08154=1024.492,-15.478,404.308,167.121,47.758,158.766
C08155=1024.498,-15.229,404.295,167.125,47.754,158.766
C08156=1024.503,-14.980,404.281,167.128,47.751,158.766
C08157=1024.510,-14.730,404.267,167.130,47.748,158.766
C08158=1024.516,-14.480,404.253,167.133,47.745,158.765
C08159=1024.522,-14.231,404.240,167.135,47.742,158.765
C08160=1024.527,-13.981,404.226,167.138,47.739,158.765
C08161=1024.534,-13.732,404.213,167.141,47.735,158.765
C08162=1024.540,-13.482,404.199,167.143,47.732,158.764
C08163=1024.546,-13.232,404.185,167.146,47.729,158.764
C08164=1024.551,-12.983,404.172,167.150,47.726,158.764
C08165=1024.558,-12.734,404.158,167.151,47.722,158.764
C08166=1024.563,-12.484,404.144,167.155,47.719,158.764
C08167=1024.570,-12.234,404.131,167.158,47.716,158.763
C08168=1024.575,-11.984,404.117,167.160,47.713,158.763
C08169=1024.582,-11.735,404.104,167.163,47.709,158.763
C08170=1024.587,-11.486,404.090,167.166,47.706,158.763
C08171=1024.594,-11.236,404.076,167.168,47.703,158.762
C08172=1024.599,-10.986,404.062,167.171,47.699,158.762
C08173=1024.606,-10.737,404.049,167.173,47.696,158.762
C08174=1024.611,-10.487,404.035,167.176,47.693,158.762
C08175=1024.618,-10.238,404.021,167.179,47.689,158.761
C08176=1024.624,-9.988,404.007,167.181,47.686,158.761
C08177=1024.630,-9.739,403.994,167.185,47.683,158.761
C08178=1024.636,-9.489,403.979,167.188,47.679,158.761
C08179=1024.642,-9.239,403.966,167.190,47.677,158.761
C08180=1024.648,-8.990,403.952,167.193,47.673,158.760
C08181=1024.654,-8.741,403.939,167.196,47.670,158.760
C08182=1024.660,-8.490,403.925,167.198,47.667,158.760
C08183=1024.666,-8.242,403.911,167.201,47.663,158.759
C08184=1024.672,-7.992,403.897,167.204,47.660,158.759
C08185=1024.679,-7.742,403.883,167.206,47.657,158.759
C08186=1024.684,-7.493,403.869,167.209,47.653,158.759
C08187=1024.690,-7.243,403.856,167.211,47.650,158.759
C08188=1024.697,-6.994,403.841,167.214,47.647,158.758
C08189=1024.703,-6.744,403.828,167.217,47.643,158.758
C08190=1024.708,-6.495,403.814,167.219,47.640,158.758
C08191=1024.715,-6.245,403.800,167.222,47.637,158.758
C08192=1024.721,-5.995,403.787,167.226,47.633,158.757
C08193=1024.728,-5.746,403.772,167.228,47.631,158.757
C08194=1024.733,-5.496,403.758,167.231,47.627,158.757
C08195=1024.740,-5.247,403.745,167.234,47.624,158.757
C08196=1024.746,-4.965,403.728,167.237,47.620,158.756
C08197=1024.754,-4.683,403.713,167.240,47.616,158.756
C08198=1024.760,-4.401,403.698,167.242,47.612,158.756
C08199=1024.768,-4.119,403.682,167.245,47.608,158.755
C08200=1024.773,-3.869,403.668,167.249,47.605,158.755
C08201=1024.780,-3.620,403.653,167.251,47.602,158.755
C08202=1024.785,-3.370,403.639,167.254,47.599,158.755
C08203=1024.791,-3.120,403.625,167.256,47.596,158.754
C08204=1024.797,-2.871,403.610,167.259,47.592,158.754
C08205=1024.802,-2.621,403.597,167.262,47.589,158.754
C08206=1024.809,-2.372,403.582,167.264,47.586,158.754
C08207=1024.815,-2.122,403.568,167.268,47.583,158.754
C08208=1024.821,-1.873,403.554,167.269,47.580,158.753
C08209=1024.827,-1.623,403.539,167.273,47.577,158.753
C08210=1024.833,-1.374,403.525,167.275,47.574,158.753
C08211=1024.839,-1.124,403.511,167.278,47.571,158.753
C08212=1024.844,-0.875,403.496,167.280,47.567,158.752
C08213=1024.851,-0.625,403.482,167.283,47.564,158.752
C08214=1024.856,-0.376,403.467,167.286,47.561,158.752
C08215=1024.863,-0.127,403.454,167.288,47.558,158.752
C08216=1024.869,0.123,403.439,167.291,47.554,158.751
C08217=1024.874,0.373,403.425,167.293,47.551,158.751
C08218=1024.881,0.622,403.410,167.297,47.548,158.751
C08219=1024.886,0.872,403.396,167.299,47.545,158.751
C08220=1024.893,1.122,403.381,167.302,47.542,158.751
C08221=1024.898,1.371,403.368,167.304,47.539,158.750
C08222=1024.905,1.621,403.353,167.307,47.536,158.750
C08223=1024.910,1.870,403.338,167.310,47.532,158.750
C08224=1024.917,2.119,403.325,167.312,47.529,158.750
C08225=1024.923,2.369,403.310,167.315,47.526,158.749
C08226=1024.928,2.618,403.296,167.317,47.522,158.749
C08227=1024.935,2.868,403.281,167.320,47.519,158.749
C08228=1024.941,3.117,403.266,167.323,47.516,158.749
C08229=1024.947,3.367,403.252,167.326,47.513,158.748
C08230=1024.952,3.616,403.238,167.328,47.510,158.748
C08231=1024.958,3.866,403.223,167.331,47.506,158.748
C08232=1024.964,4.115,403.209,167.334,47.503,158.748
C08233=1024.971,4.365,403.194,167.336,47.500,158.747
C08234=1024.977,4.615,403.180,167.339,47.497,158.747
C08235=1024.983,4.864,403.166,167.341,47.494,158.747
C08236=1024.990,5.114,403.151,167.344,47.490,158.747
C08237=1024.995,5.363,403.137,167.346,47.487,158.746
C08238=1025.001,5.613,403.122,167.350,47.484,158.746
C08239=1025.007,5.862,403.107,167.352,47.480,158.746
C08240=1025.013,6.112,403.093,167.355,47.477,158.746
C08241=1025.019,6.361,403.079,167.358,47.474,158.745
C08242=1025.026,6.611,403.064,167.360,47.471,158.745
C08243=1025.031,6.860,403.049,167.363,47.468,158.745
C08244=1025.037,7.110,403.035,167.365,47.464,158.744
C08245=1025.044,7.360,403.020,167.368,47.461,158.744
C08246=1025.050,7.608,403.006,167.371,47.458,158.744
C08247=1025.057,7.858,402.991,167.373,47.454,158.744
C08248=1025.064,8.181,402.972,167.377,47.450,158.743
C08249=1025.072,8.503,402.953,167.380,47.446,158.743
C08250=1025.080,8.826,402.934,167.383,47.442,158.743
C08251=1025.088,9.148,402.915,167.387,47.438,158.742
C08252=1025.094,9.398,402.902,167.389,47.434,158.742
C08253=1025.100,9.647,402.887,167.392,47.431,158.742
C08254=1025.106,9.897,402.872,167.394,47.427,158.741
C08255=1025.112,10.146,402.857,167.398,47.424,158.741
C08256=1025.118,10.376,402.844,167.400,47.421,158.741
C08257=1025.124,10.607,402.830,167.402,47.418,158.741
C08258=1025.130,10.837,402.817,167.405,47.415,158.741
C08259=1025.135,11.067,402.803,167.407,47.412,158.740
C08260=1025.141,11.297,402.790,167.409,47.409,158.740
C08261=1025.146,11.527,402.776,167.412,47.406,158.740
C08262=1025.152,11.757,402.763,167.415,47.403,158.740
C08263=1025.158,11.988,402.749,167.416,47.400,158.739
C08264=1025.164,12.237,402.734,167.420,47.396,158.739
C08265=1025.170,12.486,402.719,167.421,47.393,158.739
C08266=1025.177,12.736,402.704,167.425,47.390,158.738
C08267=1025.182,12.985,402.690,167.428,47.386,158.738
C08268=1025.188,13.235,402.676,167.430,47.383,158.738
C08269=1025.195,13.485,402.661,167.433,47.380,158.738
C08270=1025.201,13.734,402.646,167.435,47.377,158.737
C08271=1025.207,13.984,402.631,167.438,47.373,158.737
C08272=1025.213,14.233,402.616,167.440,47.371,158.737
C08273=1025.220,14.483,402.601,167.443,47.367,158.737
C08274=1025.226,14.732,402.587,167.445,47.364,158.736
C08275=1025.231,14.982,402.571,167.449,47.361,158.736
C08276=1025.238,15.231,402.556,167.450,47.357,158.736
C08277=1025.243,15.480,402.541,167.454,47.354,158.736
C08278=1025.250,15.729,402.526,167.456,47.351,158.735
C08279=1025.256,15.979,402.510,167.459,47.348,158.735
C08280=1025.262,16.228,402.496,167.461,47.345,158.735
C08281=1025.268,16.478,402.481,167.464,47.342,158.735
C08282=1025.274,16.728,402.466,167.466,47.338,158.734
C08283=1025.281,16.977,402.451,167.469,47.335,158.734
C08284=1025.286,17.227,402.436,167.471,47.331,158.734
C08285=1025.292,17.476,402.421,167.474,47.328,158.733
C08286=1025.298,17.726,402.406,167.476,47.326,158.733
C08287=1025.305,17.976,402.391,167.479,47.322,158.733
C08288=1025.311,18.224,402.376,167.483,47.319,158.733
C08289=1025.317,18.474,402.360,167.485,47.316,158.732
C08290=1025.323,18.723,402.345,167.488,47.312,158.732
C08291=1025.329,18.973,402.330,167.490,47.309,158.732
C08292=1025.335,19.222,402.316,167.493,47.305,158.732
C08293=1025.341,19.472,402.300,167.495,47.303,158.731
C08294=1025.347,19.721,402.284,167.498,47.299,158.731
C08295=1025.354,19.971,402.269,167.500,47.296,158.731
C08296=1025.359,20.220,402.254,167.503,47.293,158.731
C08297=1025.365,20.470,402.239,167.505,47.290,158.730
C08298=1025.371,20.720,402.224,167.507,47.286,158.730
C08299=1025.378,20.969,402.208,167.510,47.283,158.730
C08300=1025.384,21.218,402.193,167.513,47.281,158.729
C08301=1025.389,21.468,402.178,167.516,47.277,158.729
C08302=1025.396,21.717,402.162,167.518,47.274,158.729
C08303=1025.402,21.966,402.147,167.521,47.271,158.729
C08304=1025.408,22.216,402.132,167.523,47.267,158.728
C08305=1025.414,22.466,402.117,167.526,47.264,158.728
C08306=1025.420,22.714,402.102,167.528,47.261,158.728
C08307=1025.426,22.964,402.086,167.531,47.258,158.728
C08308=1025.432,23.214,402.071,167.533,47.255,158.727
C08309=1025.438,23.463,402.055,167.536,47.252,158.727
C08310=1025.445,23.713,402.040,167.538,47.248,158.727
C08311=1025.451,23.963,402.025,167.542,47.245,158.727
C08312=1025.456,24.211,402.009,167.543,47.241,158.726
C08313=1025.463,24.461,401.994,167.547,47.238,158.726
C08314=1025.468,24.711,401.979,167.549,47.236,158.726
C08315=1025.475,24.960,401.963,167.552,47.232,158.725
C08316=1025.481,25.210,401.948,167.554,47.229,158.725
C08317=1025.487,25.459,401.932,167.557,47.225,158.725
C08318=1025.494,25.709,401.917,167.559,47.222,158.725
C08319=1025.500,25.957,401.902,167.562,47.219,158.724
C08320=1025.506,26.207,401.886,167.564,47.216,158.724
C08321=1025.512,26.456,401.871,167.567,47.213,158.724
C08322=1025.518,26.706,401.855,167.569,47.209,158.723
C08323=1025.524,26.955,401.840,167.572,47.206,158.723
C08324=1025.531,27.241,401.821,167.575,47.202,158.723
C08325=1025.538,27.526,401.804,167.578,47.199,158.723
C08326=1025.545,27.811,401.786,167.581,47.195,158.722
C08327=1025.552,28.097,401.769,167.584,47.192,158.722
C08328=1025.558,28.346,401.753,167.586,47.188,158.722
C08329=1025.565,28.595,401.737,167.588,47.185,158.721
C08330=1025.570,28.845,401.721,167.592,47.182,158.721
C08331=1025.576,29.094,401.706,167.594,47.179,158.721
C08332=1025.582,29.344,401.691,167.597,47.176,158.721
C08333=1025.588,29.593,401.674,167.599,47.173,158.720
C08334=1025.594,29.843,401.659,167.602,47.169,158.720
C08335=1025.600,30.092,401.643,167.604,47.166,158.720
C08336=1025.606,30.341,401.627,167.607,47.163,158.720
C08337=1025.613,30.591,401.612,167.609,47.160,158.719
C08338=1025.619,30.840,401.596,167.611,47.157,158.719
C08339=1025.624,31.090,401.580,167.615,47.154,158.719
C08340=1025.631,31.339,401.565,167.616,47.150,158.718
C08341=1025.637,31.589,401.548,167.620,47.147,158.718
C08342=1025.642,31.839,401.533,167.622,47.144,158.718
C08343=1025.649,32.088,401.517,167.625,47.141,158.718
C08344=1025.655,32.337,401.501,167.627,47.138,158.717
C08345=1025.662,32.587,401.486,167.630,47.135,158.717
C08346=1025.667,32.835,401.470,167.632,47.131,158.717
C08347=1025.673,33.085,401.454,167.634,47.128,158.716
C08348=1025.679,33.334,401.439,167.637,47.125,158.716
C08349=1025.685,33.584,401.423,167.639,47.122,158.716
C08350=1025.691,33.833,401.406,167.643,47.119,158.716
C08351=1025.697,34.083,401.391,167.644,47.115,158.715
C08352=1025.703,34.332,401.375,167.648,47.112,158.715
C08353=1025.709,34.581,401.359,167.650,47.109,158.715
C08354=1025.716,34.831,401.344,167.653,47.105,158.715
C08355=1025.722,35.080,401.328,167.655,47.103,158.714
C08356=1025.728,35.329,401.312,167.658,47.099,158.714
C08357=1025.734,35.579,401.296,167.660,47.096,158.714
C08358=1025.740,35.829,401.280,167.663,47.092,158.713
C08359=1025.747,36.078,401.264,167.665,47.089,158.713
C08360=1025.753,36.328,401.248,167.667,47.087,158.713
C08361=1025.759,36.577,401.232,167.670,47.083,158.712
C08362=1025.766,36.827,401.217,167.673,47.080,158.712
C08363=1025.772,37.076,401.200,167.675,47.076,158.712
C08364=1025.777,37.325,401.184,167.678,47.073,158.712
C08365=1025.783,37.575,401.168,167.681,47.070,158.711
C08366=1025.789,37.824,401.152,167.683,47.067,158.711
C08367=1025.795,38.074,401.135,167.685,47.064,158.711
C08368=1025.801,38.323,401.120,167.688,47.061,158.711
C08369=1025.808,38.573,401.104,167.690,47.058,158.710
C08370=1025.814,38.822,401.088,167.693,47.054,158.710
C08371=1025.820,39.071,401.072,167.695,47.052,158.710
C08372=1025.826,39.321,401.055,167.699,47.049,158.710
C08373=1025.831,39.570,401.039,167.701,47.045,158.709
C08374=1025.837,39.819,401.023,167.703,47.042,158.709
C08375=1025.843,40.069,401.007,167.706,47.039,158.709
C08376=1025.849,40.318,400.990,167.708,47.036,158.708
C08377=1025.855,40.567,400.974,167.711,47.033,158.708
C08378=1025.862,40.816,400.958,167.713,47.029,158.708
C08379=1025.869,41.066,400.942,167.715,47.026,158.707
C08380=1025.874,41.316,400.926,167.718,47.023,158.707
C08381=1025.880,41.565,400.909,167.720,47.020,158.707
C08382=1025.886,41.814,400.893,167.724,47.017,158.707
C08383=1025.892,42.064,400.877,167.726,47.014,158.706
C08384=1025.898,42.313,400.861,167.729,47.010,158.706
C08385=1025.904,42.562,400.844,167.731,47.007,158.706
C08386=1025.910,42.812,400.828,167.733,47.004,158.706
C08387=1025.916,43.061,400.812,167.736,47.001,158.705
C08388=1025.923,43.347,400.793,167.739,46.998,158.705
C08389=1025.930,43.632,400.775,167.741,46.994,158.705
C08390=1025.936,43.917,400.756,167.744,46.990,158.704
C08391=1025.943,44.202,400.737,167.747,46.987,158.704
C08392=1025.949,44.452,400.720,167.749,46.984,158.704
C08393=1025.956,44.702,400.704,167.752,46.981,158.704
C08394=1025.962,44.950,400.687,167.755,46.978,158.703
C08395=1025.967,45.200,400.670,167.758,46.975,158.703
C08396=1025.973,45.450,400.654,167.760,46.971,158.703
C08397=1025.979,45.699,400.637,167.762,46.969,158.702
C08398=1025.985,45.948,400.621,167.765,46.966,158.702
C08399=1025.991,46.198,400.605,167.767,46.963,158.702
C08400=1025.997,46.446,400.588,167.769,46.959,158.702
C08401=1026.003,46.697,400.571,167.772,46.956,158.701
C08402=1026.009,46.946,400.554,167.775,46.953,158.701
C08403=1026.015,47.195,400.538,167.777,46.951,158.701
C08404=1026.021,47.444,400.521,167.780,46.947,158.701
C08405=1026.027,47.693,400.505,167.782,46.944,158.700
C08406=1026.032,47.943,400.488,167.785,46.941,158.700
C08407=1026.039,48.193,400.472,167.787,46.937,158.700
C08408=1026.045,48.442,400.455,167.789,46.935,158.699
C08409=1026.051,48.691,400.438,167.792,46.932,158.699
C08410=1026.057,48.941,400.422,167.794,46.928,158.699
C08411=1026.063,49.190,400.406,167.797,46.925,158.699
C08412=1026.069,49.439,400.388,167.800,46.922,158.698
C08413=1026.075,49.689,400.372,167.802,46.919,158.698
C08414=1026.081,49.938,400.355,167.805,46.916,158.698
C08415=1026.087,50.188,400.339,167.807,46.913,158.697
C08416=1026.093,50.436,400.322,167.809,46.910,158.697
C08417=1026.099,50.687,400.305,167.812,46.906,158.697
C08418=1026.105,50.936,400.289,167.814,46.904,158.697
C08419=1026.111,51.185,400.272,167.818,46.901,158.696
C08420=1026.117,51.434,400.255,167.820,46.897,158.696
C08421=1026.123,51.684,400.239,167.822,46.894,158.696
C08422=1026.129,51.933,400.221,167.825,46.891,158.695
C08423=1026.135,52.183,400.205,167.827,46.888,158.695
C08424=1026.141,52.432,400.189,167.830,46.885,158.695
C08425=1026.147,52.681,400.172,167.832,46.881,158.695
C08426=1026.154,52.931,400.155,167.834,46.878,158.694
C08427=1026.160,53.180,400.138,167.837,46.875,158.694
C08428=1026.165,53.429,400.121,167.839,46.872,158.694
C08429=1026.172,53.679,400.105,167.843,46.869,158.694
C08430=1026.178,53.928,400.088,167.845,46.865,158.693
C08431=1026.184,54.177,400.071,167.847,46.863,158.693
C08432=1026.190,54.426,400.054,167.850,46.859,158.693
C08433=1026.196,54.676,400.037,167.852,46.856,158.692
C08434=1026.202,54.926,400.021,167.855,46.853,158.692
C08435=1026.209,55.174,400.004,167.857,46.849,158.692
C08436=1026.215,55.425,399.987,167.859,46.847,158.691
C08437=1026.221,55.674,399.970,167.862,46.844,158.691
C08438=1026.227,55.923,399.954,167.864,46.840,158.691
C08439=1026.233,56.172,399.936,167.868,46.837,158.691
C08440=1026.239,56.422,399.920,167.869,46.834,158.690
C08441=1026.245,56.671,399.902,167.872,46.831,158.690
C08442=1026.251,56.920,399.886,167.875,46.828,158.690
C08443=1026.258,57.169,399.869,167.877,46.824,158.689
C08444=1026.264,57.419,399.853,167.880,46.821,158.689
C08445=1026.270,57.668,399.835,167.882,46.818,158.689
C08446=1026.276,57.918,399.818,167.885,46.815,158.688
C08447=1026.282,58.167,399.801,167.887,46.811,158.688
C08448=1026.289,58.417,399.785,167.889,46.808,158.688
C08449=1026.295,58.665,399.768,167.892,46.805,158.687
C08450=1026.300,58.915,399.751,167.894,46.802,158.687
C08451=1026.307,59.165,399.734,167.897,46.798,158.687
C08452=1026.314,59.449,399.715,167.900,46.794,158.686
C08453=1026.321,59.734,399.696,167.903,46.791,158.686
C08454=1026.328,60.019,399.677,167.905,46.787,158.686
C08455=1026.335,60.304,399.656,167.908,46.784,158.686
C08456=1026.341,60.554,399.640,167.911,46.781,158.685
C08457=1026.348,60.803,399.623,167.914,46.778,158.685
C08458=1026.354,61.052,399.606,167.916,46.774,158.685
C08459=1026.360,61.302,399.589,167.919,46.771,158.684
C08460=1026.366,61.551,399.572,167.922,46.768,158.684
C08461=1026.373,61.800,399.555,167.924,46.764,158.684
C08462=1026.379,62.049,399.538,167.927,46.761,158.683
C08463=1026.385,62.300,399.521,167.929,46.758,158.683
C08464=1026.391,62.548,399.504,167.931,46.755,158.683
C08465=1026.397,62.797,399.487,167.934,46.751,158.682
C08466=1026.404,63.047,399.470,167.936,46.748,158.682
C08467=1026.409,63.296,399.453,167.939,46.745,158.682
C08468=1026.416,63.546,399.435,167.941,46.742,158.681
C08469=1026.421,63.795,399.418,167.944,46.739,158.681
C08470=1026.428,64.045,399.401,167.946,46.735,158.681
C08471=1026.434,64.294,399.384,167.949,46.732,158.681
C08472=1026.440,64.542,399.367,167.952,46.729,158.680
C08473=1026.446,64.793,399.349,167.954,46.726,158.680
C08474=1026.452,65.041,399.332,167.956,46.723,158.680
C08475=1026.458,65.291,399.314,167.959,46.719,158.679
C08476=1026.464,65.540,399.297,167.961,46.717,158.679
C08477=1026.470,65.790,399.280,167.964,46.714,158.679
C08478=1026.476,66.039,399.263,167.966,46.710,158.678
C08479=1026.482,66.288,399.246,167.968,46.707,158.678
C08480=1026.488,66.538,399.228,167.972,46.704,158.678
C08481=1026.494,66.787,399.211,167.974,46.701,158.678
C08482=1026.500,67.036,399.193,167.977,46.698,158.677
C08483=1026.507,67.285,399.176,167.979,46.694,158.677
C08484=1026.513,67.535,399.158,167.981,46.692,158.677
C08485=1026.519,67.784,399.142,167.984,46.689,158.676
C08486=1026.525,68.034,399.124,167.986,46.685,158.676
C08487=1026.530,68.283,399.106,167.988,46.682,158.676
C08488=1026.537,68.532,399.089,167.991,46.679,158.675
C08489=1026.543,68.781,399.071,167.993,46.676,158.675
C08490=1026.549,69.031,399.053,167.997,46.673,158.675
C08491=1026.555,69.280,399.036,167.999,46.669,158.675
C08492=1026.561,69.530,399.018,168.001,46.667,158.674
C08493=1026.567,69.779,399.001,168.004,46.664,158.674
C08494=1026.574,70.028,398.984,168.006,46.660,158.674
C08495=1026.579,70.277,398.966,168.008,46.657,158.673
C08496=1026.585,70.527,398.948,168.011,46.654,158.673
C08497=1026.591,70.776,398.930,168.013,46.651,158.673
C08498=1026.598,71.025,398.913,168.017,46.648,158.673
C08499=1026.603,71.274,398.896,168.019,46.645,158.672
C08500=1026.609,71.524,398.878,168.021,46.642,158.672
C08501=1026.615,71.773,398.860,168.024,46.639,158.672
C08502=1026.622,72.023,398.843,168.026,46.636,158.671
C08503=1026.627,72.272,398.825,168.028,46.632,158.671
C08504=1026.633,72.521,398.807,168.031,46.629,158.671
C08505=1026.639,72.770,398.790,168.034,46.627,158.671
C08506=1026.646,73.020,398.772,168.036,46.623,158.670
C08507=1026.651,73.269,398.755,168.039,46.620,158.670
C08508=1026.657,73.519,398.737,168.041,46.617,158.670
C08509=1026.664,73.768,398.718,168.044,46.614,158.669
C08510=1026.669,74.017,398.701,168.046,46.611,158.669
C08511=1026.676,74.266,398.683,168.048,46.608,158.669
C08512=1026.682,74.515,398.666,168.051,46.604,158.668
C08513=1026.688,74.765,398.648,168.053,46.602,158.668
C08514=1026.693,75.014,398.630,168.056,46.598,158.668
C08515=1026.700,75.263,398.613,168.059,46.595,158.668
C08516=1026.707,75.548,398.593,168.062,46.591,158.667
C08517=1026.714,75.833,398.572,168.064,46.588,158.667
C08518=1026.721,76.118,398.552,168.067,46.584,158.666
C08519=1026.727,76.403,398.531,168.069,46.581,158.666
C08520=1026.734,76.652,398.513,168.073,46.577,158.666
C08521=1026.739,76.901,398.496,168.075,46.575,158.666
C08522=1026.745,77.150,398.477,168.078,46.571,158.665
C08523=1026.752,77.400,398.460,168.080,46.568,158.665
C08524=1026.758,77.649,398.442,168.082,46.565,158.665
C08525=1026.764,77.899,398.424,168.085,46.562,158.664
C08526=1026.770,78.148,398.406,168.087,46.559,158.664
C08527=1026.776,78.397,398.388,168.090,46.556,158.664
C08528=1026.782,78.647,398.370,168.093,46.553,158.664
C08529=1026.788,78.895,398.352,168.095,46.550,158.663
C08530=1026.793,79.145,398.333,168.097,46.547,158.663
C08531=1026.799,79.395,398.315,168.100,46.544,158.663
C08532=1026.805,79.643,398.297,168.102,46.541,158.662
C08533=1026.811,79.893,398.279,168.104,46.538,158.662
C08534=1026.817,80.142,398.262,168.108,46.535,158.662
C08535=1026.823,80.391,398.243,168.110,46.532,158.662
C08536=1026.829,80.641,398.225,168.113,46.528,158.661
C08537=1026.835,80.889,398.207,168.115,46.526,158.661
C08538=1026.841,81.139,398.189,168.117,46.523,158.661
C08539=1026.847,81.389,398.171,168.120,46.519,158.660
C08540=1026.853,81.637,398.153,168.122,46.516,158.660
C08541=1026.859,81.887,398.135,168.125,46.514,158.660
C08542=1026.866,82.137,398.117,168.128,46.510,158.659
C08543=1026.871,82.385,398.098,168.130,46.507,158.659
C08544=1026.877,82.635,398.081,168.132,46.504,158.659
C08545=1026.884,82.884,398.062,168.135,46.501,158.659
C08546=1026.889,83.133,398.044,168.137,46.498,158.658
C08547=1026.895,83.382,398.025,168.140,46.495,158.658
C08548=1026.901,83.632,398.007,168.142,46.491,158.658
C08549=1026.907,83.881,397.989,168.145,46.489,158.657
C08550=1026.913,84.130,397.971,168.148,46.486,158.657
C08551=1026.919,84.380,397.953,168.150,46.482,158.657
C08552=1026.925,84.628,397.935,168.152,46.479,158.656
C08553=1026.931,84.878,397.917,168.155,46.476,158.656
C08554=1026.938,85.127,397.898,168.157,46.473,158.656
C08555=1026.944,85.377,397.880,168.160,46.470,158.656
C08556=1026.950,85.625,397.862,168.163,46.467,158.655
C08557=1026.956,85.875,397.844,168.165,46.464,158.655
C08558=1026.962,86.124,397.825,168.168,46.461,158.655
C08559=1026.968,86.374,397.807,168.170,46.457,158.654
C08560=1026.974,86.622,397.789,168.173,46.454,158.654
C08561=1026.980,86.872,397.770,168.175,46.452,158.654
C08562=1026.986,87.122,397.752,168.177,46.448,158.653
C08563=1026.992,87.370,397.734,168.180,46.445,158.653
C08564=1026.998,87.620,397.716,168.183,46.442,158.653
C08565=1027.004,87.869,397.697,168.186,46.439,158.653
C08566=1027.010,88.119,397.679,168.188,46.436,158.652
C08567=1027.017,88.368,397.661,168.191,46.432,158.652
C08568=1027.022,88.617,397.643,168.193,46.430,158.652
C08569=1027.029,88.866,397.624,168.195,46.427,158.651
C08570=1027.035,89.115,397.606,168.198,46.423,158.651
C08571=1027.041,89.365,397.588,168.200,46.420,158.651
C08572=1027.047,89.614,397.568,168.203,46.417,158.650
C08573=1027.053,89.863,397.550,168.205,46.414,158.650
C08574=1027.059,90.112,397.532,168.208,46.411,158.650
C08575=1027.065,90.362,397.513,168.211,46.408,158.650
C08576=1027.071,90.611,397.494,168.213,46.405,158.649
C08577=1027.077,90.860,397.477,168.215,46.402,158.649
C08578=1027.082,91.109,397.458,168.218,46.399,158.649
C08579=1027.089,91.359,397.439,168.221,46.396,158.649
C08580=1027.096,91.644,397.417,168.224,46.393,158.648
C08581=1027.102,91.928,397.397,168.227,46.389,158.648
C08582=1027.109,92.213,397.375,168.229,46.385,158.647
C08583=1027.116,92.497,397.354,168.232,46.382,158.647
C08584=1027.121,92.747,397.335,168.235,46.379,158.647
C08585=1027.128,92.996,397.316,168.237,46.376,158.647
C08586=1027.134,93.246,397.297,168.240,46.373,158.646
C08587=1027.139,93.494,397.279,168.242,46.370,158.646
C08588=1027.146,93.743,397.260,168.244,46.367,158.646
C08589=1027.151,93.993,397.241,168.248,46.364,158.645
C08590=1027.158,94.242,397.223,168.250,46.361,158.645
C08591=1027.164,94.492,397.204,168.253,46.357,158.645
C08592=1027.170,94.741,397.185,168.255,46.355,158.645
C08593=1027.176,94.989,397.167,168.257,46.352,158.644
C08594=1027.181,95.239,397.148,168.260,46.348,158.644
C08595=1027.188,95.488,397.129,168.262,46.346,158.644
C08596=1027.194,95.737,397.110,168.266,46.343,158.643
C08597=1027.199,95.987,397.092,168.268,46.339,158.643
C08598=1027.206,96.236,397.073,168.270,46.336,158.643
C08599=1027.212,96.486,397.054,168.273,46.333,158.643
C08600=1027.217,96.734,397.036,168.275,46.330,158.642
C08601=1027.224,96.983,397.017,168.278,46.327,158.642
C08602=1027.229,97.233,396.998,168.280,46.324,158.642
C08603=1027.236,97.482,396.979,168.282,46.321,158.641
C08604=1027.242,97.731,396.960,168.286,46.318,158.641
C08605=1027.248,97.980,396.941,168.288,46.315,158.641
C08606=1027.254,98.229,396.923,168.291,46.311,158.640
C08607=1027.260,98.479,396.903,168.293,46.309,158.640
C08608=1027.267,98.728,396.885,168.295,46.306,158.640
C08609=1027.271,98.977,396.867,168.298,46.302,158.639
C08610=1027.278,99.227,396.848,168.301,46.300,158.639
C08611=1027.284,99.476,396.829,168.303,46.296,158.639
C08612=1027.290,99.725,396.810,168.306,46.293,158.638
C08613=1027.296,99.974,396.791,168.309,46.290,158.638
C08614=1027.302,100.223,396.771,168.311,46.287,158.638
C08615=1027.308,100.472,396.752,168.313,46.284,158.638
C08616=1027.314,100.722,396.733,168.316,46.281,158.637
C08617=1027.320,100.971,396.714,168.319,46.278,158.637
C08618=1027.326,101.220,396.695,168.321,46.276,158.637
C08619=1027.331,101.470,396.676,168.324,46.273,158.637
C08620=1027.338,101.719,396.657,168.326,46.269,158.636
C08621=1027.344,101.968,396.638,168.329,46.266,158.636
C08622=1027.349,102.218,396.619,168.332,46.263,158.636
C08623=1027.355,102.466,396.600,168.334,46.261,158.635
C08624=1027.361,102.715,396.580,168.337,46.257,158.635
C08625=1027.367,102.965,396.561,168.339,46.254,158.635
C08626=1027.373,103.214,396.543,168.342,46.251,158.635
C08627=1027.379,103.463,396.523,168.344,46.249,158.634
C08628=1027.385,103.712,396.504,168.346,46.245,158.634
C08629=1027.391,103.961,396.484,168.350,46.242,158.634
C08630=1027.397,104.210,396.465,168.352,46.239,158.633
C08631=1027.403,104.460,396.446,168.355,46.236,158.633
C08632=1027.408,104.709,396.427,168.357,46.233,158.633
C08633=1027.415,104.958,396.408,168.359,46.230,158.632
C08634=1027.421,105.207,396.388,168.363,46.227,158.632
C08635=1027.426,105.457,396.369,168.365,46.225,158.632
C08636=1027.433,105.706,396.350,168.368,46.221,158.632
C08637=1027.439,105.955,396.331,168.370,46.218,158.631
C08638=1027.445,106.204,396.311,168.372,46.215,158.631
C08639=1027.450,106.453,396.292,168.375,46.212,158.631
C08640=1027.457,106.703,396.273,168.377,46.209,158.630
C08641=1027.463,106.951,396.253,168.381,46.206,158.630
C08642=1027.468,107.201,396.234,168.383,46.203,158.630
C08643=1027.475,107.450,396.216,168.386,46.200,158.630
C08644=1027.482,107.735,396.194,168.389,46.196,158.629
C08645=1027.489,108.019,396.171,168.391,46.193,158.629
C08646=1027.496,108.304,396.149,168.394,46.190,158.629
C08647=1027.502,108.589,396.127,168.397,46.186,158.628
C08648=1027.508,108.839,396.108,168.400,46.183,158.628
C08649=1027.515,109.087,396.088,168.403,46.180,158.628
C08650=1027.521,109.337,396.069,168.405,46.177,158.627
C08651=1027.526,109.586,396.050,168.408,46.174,158.627
C08652=1027.532,109.835,396.030,168.411,46.171,158.627
C08653=1027.539,110.084,396.011,168.413,46.168,158.626
C08654=1027.545,110.333,395.991,168.415,46.165,158.626
C08655=1027.550,110.582,395.972,168.418,46.162,158.626
C08656=1027.556,110.832,395.953,168.421,46.159,158.626
C08657=1027.562,111.081,395.933,168.424,46.155,158.625
C08658=1027.568,111.330,395.914,168.426,46.153,158.625
C08659=1027.574,111.579,395.894,168.429,46.150,158.625
C08660=1027.580,111.829,395.874,168.431,46.147,158.625
C08661=1027.587,112.077,395.855,168.433,46.144,158.624
C08662=1027.592,112.327,395.835,168.437,46.141,158.624
C08663=1027.598,112.576,395.815,168.439,46.138,158.624
C08664=1027.604,112.825,395.796,168.442,46.135,158.623
C08665=1027.610,113.074,395.776,168.444,46.132,158.623
C08666=1027.616,113.323,395.757,168.448,46.129,158.623
C08667=1027.621,113.572,395.736,168.450,46.126,158.622
C08668=1027.627,113.822,395.717,168.452,46.123,158.622
C08669=1027.633,114.071,395.697,168.455,46.120,158.622
C08670=1027.639,114.319,395.677,168.457,46.117,158.622
C08671=1027.645,114.570,395.658,168.459,46.115,158.621
C08672=1027.651,114.818,395.638,168.463,46.112,158.621
C08673=1027.656,115.068,395.617,168.465,46.109,158.621
C08674=1027.662,115.317,395.598,168.468,46.106,158.621
C08675=1027.668,115.566,395.578,168.470,46.103,158.620
C08676=1027.674,115.815,395.558,168.472,46.100,158.620
C08677=1027.680,116.064,395.539,168.476,46.097,158.620
C08678=1027.686,116.313,395.519,168.478,46.094,158.620
C08679=1027.691,116.562,395.498,168.481,46.091,158.619
C08680=1027.697,116.811,395.479,168.483,46.089,158.619
C08681=1027.703,117.061,395.459,168.487,46.086,158.619
C08682=1027.709,117.310,395.439,168.489,46.083,158.619
C08683=1027.715,117.559,395.419,168.491,46.080,158.618
C08684=1027.721,117.808,395.399,168.494,46.077,158.618
C08685=1027.726,118.057,395.379,168.496,46.074,158.618
C08686=1027.732,118.306,395.359,168.500,46.071,158.617
C08687=1027.739,118.555,395.339,168.502,46.068,158.617
C08688=1027.744,118.805,395.319,168.505,46.065,158.617
C08689=1027.750,119.054,395.299,168.507,46.062,158.617
C08690=1027.756,119.303,395.279,168.510,46.060,158.616
C08691=1027.762,119.552,395.259,168.513,46.056,158.616
C08692=1027.768,119.800,395.239,168.515,46.053,158.616
C08693=1027.774,120.051,395.219,168.518,46.050,158.616
C08694=1027.780,120.299,395.199,168.520,46.048,158.615
C08695=1027.786,120.548,395.179,168.524,46.045,158.615
C08696=1027.791,120.797,395.159,168.526,46.042,158.615
C08697=1027.797,121.046,395.139,168.529,46.038,158.614
C08698=1027.803,121.296,395.119,168.531,46.036,158.614
C08699=1027.809,121.545,395.099,168.534,46.033,158.614
C08700=1027.815,121.794,395.079,168.537,46.030,158.614
C08701=1027.821,122.043,395.059,168.539,46.027,158.613
C08702=1027.827,122.292,395.039,168.542,46.024,158.613
C08703=1027.833,122.541,395.019,168.544,46.021,158.613
C08704=1027.839,122.790,394.999,168.547,46.018,158.612
C08705=1027.845,123.040,394.979,168.549,46.015,158.612
C08706=1027.850,123.289,394.959,168.553,46.012,158.612
C08707=1027.857,123.538,394.938,168.555,46.010,158.612
C08708=1027.864,123.823,394.916,168.558,46.006,158.611
C08709=1027.870,124.107,394.892,168.561,46.002,158.611
C08710=1027.878,124.392,394.870,168.564,45.999,158.611
C08711=1027.884,124.676,394.847,168.567,45.996,158.610
C08712=1027.890,124.925,394.827,168.570,45.993,158.610
C08713=1027.897,125.175,394.806,168.573,45.990,158.610
C08714=1027.903,125.423,394.786,168.576,45.987,158.609
C08715=1027.908,125.673,394.766,168.578,45.984,158.609
C08716=1027.914,125.922,394.745,168.581,45.981,158.609
C08717=1027.920,126.171,394.725,168.583,45.978,158.609
C08718=1027.926,126.420,394.705,168.587,45.975,158.608
C08719=1027.932,126.669,394.686,168.589,45.972,158.608
C08720=1027.938,126.918,394.665,168.592,45.969,158.608
C08721=1027.944,127.167,394.645,168.595,45.966,158.608
C08722=1027.950,127.416,394.625,168.597,45.963,158.607
C08723=1027.957,127.666,394.604,168.600,45.960,158.607
C08724=1027.963,127.914,394.584,168.603,45.957,158.607
C08725=1027.968,128.163,394.564,168.606,45.954,158.606
C08726=1027.975,128.413,394.544,168.608,45.951,158.606
C08727=1027.981,128.662,394.524,168.611,45.948,158.606
C08728=1027.987,128.911,394.503,168.613,45.945,158.606
C08729=1027.992,129.160,394.483,168.617,45.942,158.605
C08730=1027.998,129.409,394.463,168.619,45.939,158.605
C08731=1028.005,129.659,394.442,168.622,45.936,158.605
C08732=1028.011,129.908,394.422,168.625,45.933,158.604
C08733=1028.017,130.156,394.402,168.627,45.930,158.604
C08734=1028.023,130.406,394.382,168.631,45.927,158.604
C08735=1028.029,130.654,394.361,168.633,45.924,158.604
C08736=1028.035,130.904,394.340,168.636,45.921,158.603
C08737=1028.041,131.153,394.320,168.638,45.919,158.603
C08738=1028.046,131.402,394.299,168.642,45.916,158.603
C08739=1028.053,131.651,394.278,168.644,45.913,158.603
C08740=1028.058,131.900,394.258,168.647,45.910,158.602
C08741=1028.064,132.149,394.237,168.649,45.907,158.602
C08742=1028.070,132.399,394.217,168.652,45.904,158.602
C08743=1028.076,132.647,394.196,168.655,45.901,158.601
C08744=1028.082,132.897,394.175,168.658,45.898,158.601
C08745=1028.088,133.146,394.155,168.660,45.895,158.601
C08746=1028.094,133.395,394.135,168.663,45.893,158.601
C08747=1028.100,133.644,394.113,168.666,45.890,158.600
C08748=1028.106,133.893,394.093,168.669,45.887,158.600
C08749=1028.111,134.142,394.073,168.671,45.884,158.600
C08750=1028.117,134.391,394.051,168.674,45.881,158.600
C08751=1028.123,134.640,394.031,168.677,45.879,158.599
C08752=1028.129,134.890,394.010,168.680,45.876,158.599
C08753=1028.135,135.138,393.990,168.682,45.873,158.599
C08754=1028.141,135.388,393.969,168.685,45.869,158.599
C08755=1028.148,135.636,393.948,168.688,45.866,158.598
C08756=1028.153,135.885,393.927,168.691,45.864,158.598
C08757=1028.159,136.135,393.907,168.694,45.861,158.598
C08758=1028.165,136.383,393.886,168.696,45.858,158.598
C08759=1028.171,136.633,393.865,168.700,45.855,158.597
C08760=1028.177,136.881,393.844,168.702,45.852,158.597
C08761=1028.183,137.131,393.823,168.705,45.849,158.597
C08762=1028.188,137.380,393.803,168.707,45.847,158.597
C08763=1028.195,137.629,393.782,168.711,45.844,158.596
C08764=1028.200,137.878,393.761,168.713,45.841,158.596
C08765=1028.207,138.127,393.739,168.716,45.838,158.596
C08766=1028.213,138.376,393.720,168.719,45.835,158.596
C08767=1028.219,138.625,393.698,168.722,45.833,158.595
C08768=1028.224,138.874,393.677,168.725,45.830,158.595
C08769=1028.231,139.123,393.656,168.727,45.827,158.595
C08770=1028.236,139.372,393.636,168.730,45.824,158.595
C08771=1028.242,139.622,393.614,168.733,45.821,158.594
C08772=1028.249,139.906,393.590,168.736,45.818,158.594
C08773=1028.255,140.190,393.567,168.739,45.815,158.594
C08774=1028.261,140.475,393.542,168.742,45.812,158.594
C08775=1028.269,140.760,393.518,168.746,45.808,158.593
C08776=1028.274,141.008,393.497,168.748,45.805,158.593
C08777=1028.281,141.258,393.476,168.752,45.802,158.593
C08778=1028.286,141.506,393.455,168.754,45.800,158.592
C08779=1028.293,141.755,393.433,168.757,45.797,158.592
C08780=1028.298,142.004,393.413,168.759,45.794,158.592
C08781=1028.304,142.254,393.391,168.763,45.791,158.592
C08782=1028.309,142.503,393.371,168.766,45.788,158.591
C08783=1028.316,142.752,393.350,168.768,45.786,158.591
C08784=1028.322,143.000,393.328,168.772,45.783,158.591
C08785=1028.328,143.250,393.307,168.774,45.780,158.591
C08786=1028.334,143.499,393.286,168.777,45.777,158.590
C08787=1028.339,143.748,393.264,168.779,45.774,158.590
C08788=1028.346,143.997,393.243,168.783,45.771,158.590
C08789=1028.352,144.246,393.223,168.786,45.768,158.590
C08790=1028.358,144.495,393.201,168.788,45.766,158.589
C08791=1028.363,144.743,393.180,168.791,45.763,158.589
C08792=1028.369,144.993,393.158,168.794,45.760,158.589
C08793=1028.375,145.242,393.137,168.797,45.757,158.589
C08794=1028.381,145.491,393.116,168.800,45.754,158.588
C08795=1028.388,145.740,393.095,168.802,45.752,158.588
C08796=1028.393,145.988,393.074,168.806,45.749,158.588
C08797=1028.399,146.238,393.053,168.809,45.746,158.588
C08798=1028.405,146.487,393.031,168.811,45.743,158.587
C08799=1028.411,146.736,393.010,168.814,45.740,158.587
C08800=1028.417,146.985,392.988,168.817,45.738,158.587
C08801=1028.423,147.234,392.967,168.820,45.735,158.587
C08802=1028.429,147.483,392.945,168.824,45.732,158.587
C08803=1028.435,147.733,392.925,168.826,45.730,158.586
C08804=1028.440,147.981,392.903,168.829,45.727,158.586
C08805=1028.446,148.230,392.882,168.831,45.724,158.586
C08806=1028.453,148.480,392.860,168.835,45.721,158.586
C08807=1028.458,148.728,392.839,168.838,45.718,158.585
C08808=1028.464,148.977,392.817,168.840,45.716,158.585
C08809=1028.470,149.226,392.796,168.843,45.713,158.585
C08810=1028.476,149.475,392.774,168.846,45.710,158.585
C08811=1028.482,149.724,392.753,168.849,45.708,158.585
C08812=1028.487,149.973,392.731,168.852,45.705,158.584
C08813=1028.493,150.222,392.709,168.855,45.702,158.584
C08814=1028.499,150.471,392.687,168.858,45.699,158.584
C08815=1028.505,150.720,392.666,168.860,45.696,158.584
C08816=1028.511,150.969,392.645,168.863,45.694,158.583
C08817=1028.517,151.218,392.623,168.867,45.691,158.583
C08818=1028.523,151.467,392.602,168.869,45.688,158.583
C08819=1028.529,151.716,392.580,168.873,45.686,158.583
C08820=1028.535,151.965,392.558,168.876,45.683,158.582
C08821=1028.540,152.214,392.536,168.878,45.680,158.582
C08822=1028.546,152.463,392.515,168.881,45.677,158.582
C08823=1028.552,152.712,392.493,168.885,45.674,158.582
C08824=1028.558,152.962,392.472,168.887,45.672,158.581
C08825=1028.564,153.210,392.450,168.890,45.669,158.581
C08826=1028.570,153.459,392.428,168.893,45.666,158.581
C08827=1028.577,153.708,392.406,168.896,45.664,158.581
C08828=1028.581,153.957,392.384,168.899,45.661,158.581
C08829=1028.588,154.206,392.363,168.902,45.658,158.580
C08830=1028.594,154.455,392.341,168.905,45.655,158.580
C08831=1028.600,154.704,392.320,168.908,45.652,158.580
C08832=1028.605,154.953,392.297,168.910,45.650,158.580
C08833=1028.611,155.202,392.275,168.914,45.647,158.580
C08834=1028.617,155.451,392.254,168.917,45.645,158.579
C08835=1028.623,155.700,392.232,168.919,45.642,158.579
C08836=1028.630,155.984,392.207,168.924,45.639,158.579
C08837=1028.636,156.269,392.182,168.927,45.636,158.579
C08838=1028.643,156.552,392.157,168.930,45.632,158.578
C08839=1028.650,156.836,392.132,168.933,45.629,158.578
C08840=1028.656,157.085,392.110,168.936,45.626,158.578
C08841=1028.662,157.335,392.088,168.940,45.624,158.578
C08842=1028.668,157.583,392.066,168.942,45.622,158.577
C08843=1028.674,157.833,392.044,168.946,45.619,158.577
C08844=1028.679,158.081,392.023,168.949,45.616,158.577
C08845=1028.686,158.330,392.001,168.951,45.613,158.577
C08846=1028.691,158.579,391.978,168.955,45.611,158.577
C08847=1028.697,158.828,391.956,168.958,45.608,158.576
C08848=1028.704,159.078,391.935,168.960,45.605,158.576
C08849=1028.710,159.326,391.913,168.963,45.602,158.576
C08850=1028.715,159.575,391.891,168.967,45.599,158.576
C08851=1028.721,159.824,391.868,168.969,45.597,158.576
C08852=1028.727,160.073,391.846,168.972,45.595,158.575
C08853=1028.733,160.322,391.823,168.976,45.592,158.575
C08854=1028.737,160.571,391.801,168.978,45.590,158.575
C08855=1028.744,160.819,391.779,168.982,45.587,158.575
C08856=1028.749,161.069,391.757,168.985,45.584,158.575
C08857=1028.755,161.318,391.734,168.987,45.582,158.574
C08858=1028.760,161.567,391.711,168.991,45.580,158.574
C08859=1028.766,161.815,391.689,168.994,45.577,158.574
C08860=1028.772,162.064,391.666,168.997,45.575,158.574
C08861=1028.777,162.314,391.644,169.000,45.572,158.574
C08862=1028.784,162.562,391.622,169.003,45.569,158.573
C08863=1028.789,162.812,391.600,169.006,45.567,158.573
C08864=1028.794,163.060,391.577,169.009,45.564,158.573
C08865=1028.800,163.309,391.554,169.013,45.562,158.573
C08866=1028.806,163.558,391.533,169.015,45.559,158.573
C08867=1028.812,163.807,391.510,169.018,45.556,158.572
C08868=1028.818,164.056,391.487,169.022,45.554,158.572
C08869=1028.824,164.305,391.465,169.024,45.551,158.572
C08870=1028.830,164.554,391.442,169.027,45.549,158.572
C08871=1028.835,164.802,391.419,169.031,45.546,158.572
C08872=1028.840,165.052,391.397,169.033,45.544,158.572
C08873=1028.847,165.300,391.375,169.037,45.541,158.571
C08874=1028.852,165.549,391.352,169.040,45.538,158.571
C08875=1028.858,165.799,391.330,169.043,45.536,158.571
C08876=1028.864,166.048,391.307,169.046,45.533,158.571
C08877=1028.870,166.296,391.284,169.049,45.531,158.571
C08878=1028.876,166.545,391.261,169.052,45.528,158.571
C08879=1028.881,166.795,391.239,169.055,45.526,158.570
C08880=1028.888,167.043,391.217,169.058,45.523,158.570
C08881=1028.893,167.291,391.194,169.062,45.521,158.570
C08882=1028.899,167.540,391.171,169.065,45.518,158.570
C08883=1028.904,167.790,391.149,169.067,45.516,158.570
C08884=1028.910,168.038,391.127,169.071,45.513,158.570
C08885=1028.916,168.287,391.104,169.074,45.511,158.569
C08886=1028.922,168.536,391.081,169.077,45.508,158.569
C08887=1028.928,168.785,391.058,169.080,45.506,158.569
C08888=1028.934,169.034,391.036,169.083,45.503,158.569
C08889=1028.940,169.283,391.013,169.087,45.501,158.569
C08890=1028.945,169.532,390.990,169.090,45.498,158.568
C08891=1028.951,169.781,390.967,169.093,45.496,158.568
C08892=1028.958,170.030,390.945,169.096,45.493,158.568
C08893=1028.963,170.278,390.922,169.099,45.490,158.568
C08894=1028.969,170.527,390.899,169.103,45.488,158.568
C08895=1028.975,170.776,390.876,169.106,45.485,158.567
C08896=1028.981,171.025,390.855,169.109,45.483,158.567
C08897=1028.987,171.274,390.832,169.112,45.480,158.567
C08898=1028.992,171.523,390.809,169.115,45.478,158.567
C08899=1028.998,171.772,390.786,169.119,45.475,158.567
C08900=1029.005,172.056,390.759,169.122,45.472,158.567
C08901=1029.012,172.340,390.734,169.125,45.469,158.566
C08902=1029.019,172.624,390.708,169.129,45.466,158.566
C08903=1029.025,172.907,390.682,169.133,45.463,158.566
C08904=1029.031,173.156,390.659,169.136,45.461,158.566
C08905=1029.038,173.404,390.636,169.140,45.458,158.566
C08906=1029.043,173.653,390.613,169.143,45.456,158.566
C08907=1029.050,173.903,390.590,169.145,45.453,158.565
C08908=1029.055,174.152,390.567,169.149,45.451,158.565
C08909=1029.062,174.400,390.545,169.152,45.448,158.565
C08910=1029.068,174.649,390.522,169.156,45.446,158.565
C08911=1029.073,174.898,390.499,169.159,45.443,158.565
C08912=1029.079,175.147,390.476,169.162,45.440,158.564
C08913=1029.085,175.396,390.453,169.165,45.438,158.564
C08914=1029.091,175.644,390.431,169.168,45.435,158.564
C08915=1029.097,175.893,390.408,169.172,45.433,158.564
C08916=1029.103,176.143,390.384,169.175,45.430,158.564
C08917=1029.109,176.392,390.361,169.179,45.428,158.564
C08918=1029.115,176.640,390.339,169.182,45.425,158.563
C08919=1029.121,176.889,390.316,169.185,45.423,158.563
C08920=1029.127,177.137,390.293,169.189,45.420,158.563
C08921=1029.133,177.386,390.270,169.191,45.418,158.563
C08922=1029.139,177.636,390.246,169.194,45.415,158.563
C08923=1029.146,177.885,390.224,169.198,45.412,158.562
C08924=1029.151,178.133,390.201,169.201,45.410,158.562
C08925=1029.157,178.382,390.178,169.205,45.407,158.562
C08926=1029.163,178.631,390.154,169.208,45.405,158.562
C08927=1029.170,178.880,390.131,169.211,45.402,158.562
C08928=1029.176,179.129,390.109,169.215,45.400,158.562
C08929=1029.182,179.378,390.086,169.218,45.397,158.561
C08930=1029.187,179.627,390.063,169.222,45.394,158.561
C08931=1029.194,179.876,390.039,169.225,45.392,158.561
C08932=1029.200,180.124,390.016,169.228,45.390,158.561
C08933=1029.206,180.373,389.993,169.231,45.387,158.561
C08934=1029.212,180.622,389.971,169.234,45.385,158.561
C08935=1029.219,180.871,389.947,169.238,45.382,158.560
C08936=1029.224,181.120,389.924,169.241,45.379,158.560
C08937=1029.230,181.369,389.901,169.244,45.377,158.560
C08938=1029.237,181.617,389.878,169.248,45.374,158.560
C08939=1029.243,181.866,389.854,169.251,45.371,158.560
C08940=1029.249,182.115,389.831,169.255,45.369,158.560
C08941=1029.255,182.364,389.808,169.258,45.366,158.560
C08942=1029.261,182.613,389.784,169.262,45.364,158.559
C08943=1029.268,182.862,389.762,169.265,45.361,158.559
C08944=1029.273,183.110,389.738,169.268,45.359,158.559
C08945=1029.279,183.359,389.715,169.272,45.357,158.559
C08946=1029.284,183.608,389.691,169.276,45.355,158.559
C08947=1029.290,183.857,389.667,169.278,45.352,158.559
C08948=1029.297,184.106,389.644,169.281,45.350,158.559
C08949=1029.302,184.354,389.619,169.285,45.348,158.559
C08950=1029.308,184.603,389.596,169.288,45.345,158.558
C08951=1029.313,184.852,389.572,169.292,45.343,158.558
C08952=1029.320,185.101,389.548,169.296,45.341,158.558
C08953=1029.325,185.350,389.525,169.299,45.338,158.558
C08954=1029.331,185.598,389.501,169.302,45.336,158.558
C08955=1029.337,185.848,389.478,169.305,45.334,158.558
C08956=1029.342,186.096,389.453,169.308,45.332,158.558
C08957=1029.348,186.345,389.430,169.312,45.329,158.558
C08958=1029.354,186.594,389.405,169.315,45.327,158.557
C08959=1029.360,186.843,389.382,169.319,45.324,158.557
C08960=1029.366,187.091,389.358,169.322,45.322,158.557
C08961=1029.371,187.340,389.334,169.326,45.320,158.557
C08962=1029.377,187.589,389.311,169.329,45.318,158.557
C08963=1029.383,187.838,389.287,169.333,45.316,158.557
C08964=1029.390,188.121,389.259,169.336,45.313,158.557
C08965=1029.396,188.404,389.232,169.341,45.310,158.557
C08966=1029.403,188.688,389.205,169.344,45.307,158.556
C08967=1029.410,188.971,389.178,169.349,45.305,158.556
C08968=1029.416,189.220,389.154,169.352,45.303,158.556
C08969=1029.422,189.468,389.130,169.356,45.301,158.556
C08970=1029.427,189.718,389.106,169.359,45.298,158.556
C08971=1029.433,189.966,389.083,169.363,45.295,158.556
C08972=1029.439,190.215,389.058,169.366,45.293,158.556
C08973=1029.445,190.464,389.034,169.370,45.291,158.556
C08974=1029.451,190.712,389.010,169.373,45.289,158.556
C08975=1029.457,190.961,388.986,169.376,45.287,158.556
C08976=1029.463,191.210,388.962,169.379,45.285,158.555
C08977=1029.469,191.459,388.938,169.383,45.282,158.555
C08978=1029.475,191.708,388.915,169.386,45.280,158.555
C08979=1029.480,191.956,388.890,169.390,45.277,158.555
C08980=1029.487,192.205,388.866,169.393,45.275,158.555
C08981=1029.492,192.454,388.842,169.397,45.273,158.555
C08982=1029.499,192.703,388.818,169.400,45.271,158.555
C08983=1029.505,192.951,388.795,169.405,45.268,158.555
C08984=1029.511,193.200,388.770,169.408,45.266,158.555
C08985=1029.517,193.449,388.746,169.412,45.264,158.555
C08986=1029.523,193.698,388.722,169.416,45.262,158.555
C08987=1029.529,193.946,388.698,169.419,45.260,158.554
C08988=1029.535,194.196,388.673,169.422,45.257,158.554
C08989=1029.541,194.444,388.650,169.426,45.255,158.554
C08990=1029.547,194.693,388.625,169.429,45.252,158.554
C08991=1029.553,194.941,388.601,169.433,45.250,158.554
C08992=1029.558,195.191,388.577,169.437,45.248,158.554
C08993=1029.565,195.439,388.553,169.440,45.246,158.554
C08994=1029.570,195.688,388.528,169.444,45.244,158.554
C08995=1029.576,195.937,388.505,169.447,45.241,158.554
C08996=1029.583,196.186,388.481,169.451,45.239,158.554
C08997=1029.589,196.434,388.456,169.454,45.237,158.553
C08998=1029.595,196.682,388.432,169.458,45.235,158.553
C08999=1029.601,196.932,388.407,169.461,45.233,158.553
C09000=1029.607,197.180,388.383,169.465,45.230,158.553
C09001=1029.613,197.429,388.359,169.470,45.228,158.553
C09002=1029.619,197.678,388.335,169.473,45.225,158.553
C09003=1029.625,197.927,388.311,169.476,45.223,158.553
C09004=1029.632,198.175,388.286,169.480,45.221,158.553
C09005=1029.637,198.424,388.262,169.483,45.218,158.553
C09006=1029.644,198.673,388.238,169.487,45.216,158.553
C09007=1029.649,198.921,388.213,169.491,45.214,158.552
C09008=1029.656,199.170,388.189,169.494,45.212,158.552
C09009=1029.662,199.419,388.164,169.498,45.210,158.552
C09010=1029.668,199.667,388.140,169.502,45.207,158.552
C09011=1029.674,199.917,388.116,169.506,45.205,158.552
C09012=1029.681,200.166,388.092,169.509,45.203,158.552
C09013=1029.686,200.414,388.067,169.513,45.201,158.552
C09014=1029.692,200.663,388.042,169.516,45.198,158.552
C09015=1029.699,200.912,388.018,169.520,45.197,158.552
C09016=1029.704,201.160,387.993,169.524,45.195,158.552
C09017=1029.710,201.409,387.968,169.527,45.193,158.552
C09018=1029.717,201.658,387.943,169.531,45.190,158.552
C09019=1029.722,201.906,387.919,169.535,45.188,158.552
C09020=1029.728,202.155,387.893,169.539,45.186,158.552
C09021=1029.734,202.403,387.870,169.543,45.184,158.552
C09022=1029.740,202.652,387.844,169.546,45.182,158.552
C09023=1029.746,202.901,387.820,169.550,45.180,158.551
C09024=1029.752,203.149,387.795,169.553,45.178,158.551
C09025=1029.758,203.399,387.770,169.557,45.175,158.551
C09026=1029.764,203.647,387.745,169.561,45.174,158.551
C09027=1029.771,203.896,387.721,169.565,45.171,158.551
C09028=1029.795,204.944,387.616,169.926,45.275,158.610
C09029=1029.806,205.313,387.577,169.931,45.273,158.610
C09030=1029.816,205.682,387.538,169.934,45.271,158.610
C09031=1029.826,206.051,387.500,169.938,45.270,158.610
C09032=1029.835,206.421,387.461,169.942,45.267,158.610
C09033=1029.842,206.669,387.434,169.945,45.266,158.610
C09034=1029.849,206.917,387.408,169.948,45.264,158.610
C09035=1029.856,207.166,387.382,169.951,45.263,158.610
C09036=1029.862,207.415,387.355,169.954,45.262,158.610
C09037=1029.869,207.663,387.329,169.956,45.261,158.610
C09038=1029.875,207.911,387.303,169.959,45.259,158.610
C09039=1029.883,208.160,387.276,169.962,45.259,158.610
C09040=1029.889,208.408,387.250,169.964,45.257,158.610
C09041=1029.895,208.657,387.223,169.967,45.256,158.610
C09042=1029.903,208.906,387.197,169.969,45.255,158.610
C09043=1029.909,209.154,387.171,169.972,45.253,158.610
C09044=1029.916,209.403,387.144,169.975,45.252,158.610
C09045=1029.922,209.651,387.118,169.978,45.251,158.610
C09046=1029.929,209.900,387.091,169.981,45.249,158.610
C09047=1029.936,210.148,387.065,169.983,45.248,158.610
C09048=1029.942,210.397,387.038,169.986,45.247,158.610
C09049=1029.949,210.646,387.012,169.989,45.245,158.610
C09050=1029.956,210.893,386.985,169.992,45.245,158.610
C09051=1029.962,211.142,386.958,169.995,45.243,158.610
C09052=1029.969,211.390,386.932,169.998,45.242,158.610
C09053=1029.975,211.639,386.905,170.000,45.241,158.610
C09054=1029.982,211.888,386.878,170.003,45.240,158.610
C09055=1029.989,212.136,386.852,170.006,45.239,158.611
C09056=1029.995,212.385,386.825,170.009,45.238,158.611
C09057=1030.002,212.633,386.799,170.012,45.236,158.611
C09058=1030.008,212.882,386.772,170.014,45.235,158.611
C09059=1030.015,213.130,386.745,170.017,45.234,158.611
C09060=1030.021,213.379,386.719,170.020,45.233,158.611
C09061=1030.029,213.627,386.691,170.023,45.232,158.611
C09062=1030.035,213.876,386.664,170.026,45.230,158.611
C09063=1030.042,214.124,386.638,170.029,45.229,158.611
C09064=1030.048,214.373,386.611,170.032,45.228,158.611
C09065=1030.055,214.621,386.584,170.034,45.227,158.611
C09066=1030.062,214.869,386.558,170.037,45.226,158.611
C09067=1030.068,215.118,386.531,170.040,45.224,158.611
C09068=1030.076,215.366,386.504,170.043,45.223,158.611
C09069=1030.081,215.615,386.477,170.046,45.222,158.611
C09070=1030.089,215.864,386.451,170.049,45.221,158.611
C09071=1030.095,216.112,386.423,170.051,45.220,158.611
C09072=1030.102,216.360,386.397,170.054,45.218,158.611
C09073=1030.108,216.609,386.370,170.057,45.218,158.611
C09074=1030.116,216.857,386.343,170.060,45.216,158.611
C09075=1030.121,217.106,386.316,170.063,45.215,158.611
C09076=1030.128,217.354,386.290,170.066,45.214,158.611
C09077=1030.135,217.603,386.262,170.069,45.213,158.612
C09078=1030.142,217.852,386.236,170.071,45.212,158.612
C09079=1030.148,218.100,386.209,170.074,45.210,158.612
C09080=1030.155,218.348,386.182,170.077,45.209,158.612
C09081=1030.162,218.597,386.155,170.080,45.208,158.612
C09082=1030.169,218.845,386.128,170.083,45.207,158.612
C09083=1030.176,219.093,386.102,170.086,45.206,158.612
C09084=1030.182,219.342,386.074,170.088,45.204,158.612
C09085=1030.193,219.717,386.033,170.093,45.203,158.612
C09086=1030.202,220.092,385.992,170.097,45.202,158.612
C09087=1030.213,220.467,385.951,170.102,45.200,158.612
C09088=1030.222,220.842,385.910,170.106,45.198,158.612
C09089=1030.229,221.090,385.883,170.109,45.197,158.612
C09090=1030.235,221.339,385.856,170.112,45.196,158.612
C09091=1030.242,221.587,385.828,170.114,45.195,158.612
C09092=1030.248,221.835,385.801,170.117,45.194,158.612
C09093=1030.255,222.084,385.775,170.120,45.193,158.613
C09094=1030.262,222.332,385.747,170.123,45.192,158.613
C09095=1030.268,222.581,385.720,170.126,45.191,158.613
C09096=1030.275,222.830,385.692,170.129,45.190,158.613
C09097=1030.281,223.077,385.665,170.132,45.188,158.613
C09098=1030.288,223.326,385.638,170.136,45.188,158.613
C09099=1030.295,223.575,385.611,170.138,45.186,158.613
C09100=1030.301,223.823,385.583,170.141,45.186,158.613
C09101=1030.308,224.071,385.555,170.144,45.184,158.613
C09102=1030.315,224.320,385.529,170.147,45.184,158.613
C09103=1030.321,224.568,385.501,170.150,45.182,158.613
